(* CODESYS project sensata_laser.library
   Company: Sensata Technologies
   DocFormat: reStructuredText
   Description: This library is for the Laser devices
   Version: 1.0.1
   Placeholder: Sensata_Laser
   Title: Sensata_Laser

Project tree, tasks and I/O mapping:
  libraries: Sensata_Common, * (Sensata Technologies); Sensata_Utilities, * (Sensata Technologies); Tc2_Standard, * (Beckhoff Automation GmbH); Tc2_System, * (Beckhoff Automation GmbH); Tc2_Utilities, * (Beckhoff Automation GmbH); Tc3_Module, * (Beckhoff Automation GmbH)
  Abstract/
    function block FB_Laser [ST]: M_GetLaserStatus, M_LaserOff, M_LaserOn, P_bLaserControlBusy, P_bLaserOn
    function block FB_LaserMarker [ST]: M_SendMarkingParams_BlockRange, M_StartMarking, M_StopMarking, M_UpdateAllMarkingInformation, M_UpdateSingleBlockMarkingInformation, M_GetLaserStatus
    function block FB_LaserScanner [ST]: M_Trigger
  Concrete/
    IPG/
      function block FB_IPGD30 [ST]: M_Abort, P_bAbortBusy, M_Connect, M_Disconnect, M_GetConnectStatus, P_bConnectBusy, P_bConnected, M_Disable, M_Enable, M_GetEnableStatus, P_bEnableBusy, P_bEnabled, M_GetPowerStatus, M_PowerOff, M_PowerOn, P_bPowerBusy, P_bPoweredOn, M_GetCurrentProgram, M_GetProgramState, M_LoadProgram, M_PauseProgram, M_StartProgram, M_StopProgram, P_bProgramControlBusy, P_enumProgramState, P_strCurrentProgram, M_Reset, P_bResetBusy, A_CommandRecovery, M_RouterHelper
      function block FB_IPGWeld [ST]: M_Abort, P_bAbortBusy, M_Connect, M_Disconnect, M_GetConnectStatus, P_bConnectBusy, P_bConnected, M_Disable, M_Enable, M_GetEnableStatus, P_bEnableBusy, P_bEnabled, M_GetPowerStatus, M_PowerOff, M_PowerOn, P_bPowerBusy, P_bPoweredOn, M_GetCurrentProgram, M_GetProgramState, M_LoadProgram, M_PauseProgram, M_StartProgram, M_StopProgram, P_bProgramControlBusy, P_enumProgramState, P_strCurrentProgram, M_Reset, P_bResetBusy, M_Trigger, A_CommandRecovery, M_CommandTemplate, M_RouterHelper
    Keyence MDX-2000/
      function block FB_KeyenceLaserMarkerMDX2000 [LD]: M_Connect, M_Disconnect, M_GetConnectStatus, P_bConnectBusy, P_bConnected, M_PeakCurrentProgram, M_SendMarkingParams_BlockRange, M_StartMarking, M_StopMarking, M_UpdateAllMarkingInformation, M_UpdateSingleBlockMarkingInformation, M_GetCurrentProgram, M_GetProgramState, M_LoadProgram, M_PauseProgram, M_SaveCurrentLaserProgramtoPC, M_SendProgramtoLaser, M_StartProgram, M_StopProgram, M_UpdateSingleProgramBlockData, M_UpdateSingleProgramBlockMarkEnabled, P_bProgramControlBusy, P_enumProgramState, P_strCurrentProgram, M_GetLaserActivatedStatus, M_GetLaserErrorStatus, M_GetLaserMarkingStatus, M_GetLaserStatus, M_Reset, P_bResetBusy, A_CommandRecovery, M_RouterHelper
      data type KeyenceLaserMarkerMDX2000_Error
  DUTs/
    data type BlockTypes
    data type OneBlockInfo
  Interfaces/
    interface I_LaserControl: M_GetLaserStatus, M_LaserOff, M_LaserOn, P_bLaserControlBusy, P_bLaserOn
    interface I_Markable: M_StartMarking, M_StopMarking, M_UpdateAllMarkingInformation, M_UpdateSingleBlockMarkingInformation
    interface I_Triggerable: M_Trigger
  Project Information/
    function F_GetCompany [ST]
    function F_GetTitle [ST]
    function F_GetVersion [ST]
  Version/
    global variables Global_Version
  global variables GVL_LaserMarker
*)

// Concrete/Keyence MDX-2000/KeyenceLaserMarkerMDX2000_Error
{attribute 'qualified_only'}
{attribute 'strict'}
TYPE KeyenceLaserMarkerMDX2000_Error :
(
	None := 0,
	
	CommandRouterError							:= 0100, 		// Error on the command router FB
	CommandFault 								:= 0101, 		// Command failed to execute
	                            				         		
	FailedToConnect 							:= 0200, 		// Connect command failed
	FailedToDisconnect 							:= 0201, 		// Disonnect command failed
	FailedToGetConnectStatus 					:= 0202, 		// GetConnectStatus command failed
	                                                     		
	FailedToPeakCurrentProgram  				:= 0300, 		// Failed to Peak Current Program 
	FailedToSaveCurrentLaserProgramToPC 		:= 0301, 		//Failed to Save Current Laser Program to PC
	FailedToSendProgramToLaser					:= 0302, 		// Failed to Send Program To Laser
	FailedToStartMarking						:= 0303, 		// Laser Failed to Start Marking
	FailedToStopMarking							:= 0304, 		// Laser Failed to Stop Marking
	FailedToLoadProgram							:= 0310, 		// LoadProgram command failed
	FailedToGetCurrentProgram					:= 0311, 		// GetCurrentProgram command failed
	FailedToStartProgram						:= 0312, 		// StartProgram command failed
	FailedToStopProgram							:= 0313, 		// StopProgram command failed
	FailedToPauseProgram						:= 0314, 		// PauseProgram command failed
	FailedToGetProgramState						:= 0315, 		// GetProgramState command failed
	FailedToGetLaserStatus						:= 0316, 		// GetLaserStatus command failed
	FailedToGetLaserErrorStatus 				:= 0317, 		// GetLaserErrorStatus command failed
	FailedToGetLaserMarkingStatus 				:= 0318, 		// GetLaserMarkingStatus command failed
	FailedToGetLaserActivatedStatus				:= 0319, 		// GetLaserActivatedStatus command failed
	FailedToUpdateSingleBlockMarkEnabledProperty := 0320,		// UpdateSingleBlockMarkEnabled command failed
	FailedToUpdateSingleBlockData				:= 0321,		// UpdateSingleBlockData command failed
	FailedToUpdateAllMarkingInformation			:= 0322,		// UpdateAllMarkingInformation command failed
	FailedToUpdateSingleBlockMarkingInformation := 0323,		// UpdateSingleBlockMarkingInformation command failed
	FailedToGetPartLimitsFromDB					:= 0324,		// GetPartLimitsFromDB command failed
	FailedToSendMarkingParams_BlockRange        := 0325,		// SendMarkingParams_BlockRange command failed
                                                     		
	FailedToEnable								:= 0400, 		// Enable command failed
	FailedToDisable								:= 0401, 		// Disable command failed
	FailedToGetEnableStatus						:= 0402, 		// GetEnableStatus command failed
	                            				         		
	FailedToPowerOn								:= 0500, 		// PowerOn command failed
	FailedToPowerOff							:= 0501, 		// PowerOff command failed
	FailedToGetPowerStatus						:= 0502, 		// GetPowerStatus command failed
	                            				         		
	FailedToReset								:= 0600, 		// Reset command failed
	FailedToClearLaserErrors					:= 0601, 		// Failed to Clear Laser Errors
                                				         		
	FailedToGetSafetyStatus						:= 0700, 		// GetSafetyStatus command failed
	RobotSafetyFault							:= 0701  		// Robot safety fault occurred
) UDINT;
END_TYPE

// DUTs/BlockTypes
{attribute 'qualified_only'}
{attribute 'strict'}
TYPE BlockTypes :
(
  BLOCK_CHARACTER:=0, 
  BLOCK_RESERVED1:=1, 
  BLOCK_BARCODE:=2, 
  BLOCK_GS1DATABAR:=3, 
  BLOCK_2DCODE:=4, 
  BLOCK_RESERVED2:=5, 
  BLOCK_LOGO:=6, 
  BLOCK_PHOTO:=7, 
  BLOCK_PROCESSING:=8, 
  BLOCK_RESERVED3:=9
)INT;
END_TYPE

// DUTs/OneBlockInfo
TYPE OneBlockInfo :
STRUCT
	MarkEnabled : BOOL;
	BlockText : T_MaxString;
END_STRUCT
END_TYPE

// Version/Global_Version
{attribute 'TcGenerated'}
{attribute 'no-analysis'}
{attribute 'linkalways'}
// This function has been automatically generated from the project information.
VAR_GLOBAL CONSTANT
	{attribute 'const_non_replaced'}
	stLibVersion_Sensata_Laser : ST_LibVersion := (iMajor := 1, iMinor := 0, iBuild := 1, iRevision := 0, nFlags := 0, sVersion := '1.0.1');
END_VAR

// GVL_LaserMarker
VAR_GLOBAL
	LaserConnected : BOOL := FALSE;
	LaserDisconnected : BOOL := FALSE;
	LaserMarkerErrorsCleared : BOOL := FALSE;
	UpdateAllBlocksInLaserProgramSuccess : BOOL := FALSE;
	UpdateSingleBlockInLaserProgramSuccess : BOOL := FALSE;
	UpdateSingleBlockMarkEnabledSuccess : BOOL := FALSE;
	PeakCurrentProgramSuccess : BOOL := FALSE;
	SendProgramToLaserSuccess : BOOL := FALSE;
	SaveCurrentLaserProgramToPCSuccess : BOOL := FALSE;
	StartMarkingSuccess : BOOL := FALSE;
	StopMarkingSuccess : BOOL := FALSE;
	_bIsLaserActivated : BOOL := FALSE;
	_bIsLaserError : BOOL := FALSE;
	_bIsLaserMarking : BOOL := FALSE;
	KeyenceLaserProgramFolder : STRING := 'C:\MSDCommon\MarkingFiles\Program';
	KeyenceLaserModel : STRING := 'MARKINGUNIT_MDX2520';//For Marker Builder Plus and HVC(APT inline Cal #31) DAGZ181089
	KeyenceLaserIPAddress : STRING := '127.0.0.1';

END_VAR

// Abstract/FB_Laser
FUNCTION_BLOCK FB_Laser EXTENDS FB_Device IMPLEMENTS
I_LaserControl
VAR_INPUT
END_VAR
VAR_OUTPUT
END_VAR
VAR
	dev_bLaserOn: BOOL; // TRUE if the laser is on
END_VAR


METHOD M_GetLaserStatus : BOOL
VAR_OUTPUT
	(* TRUE if the laser is on, FALSE otherwise. *)
	bLaserOn	: BOOL;
END_VAR
bLaserOn:=dev_bLaserOn;
M_GetLaserStatus:=TRUE;
END_METHOD

(*Turn off Laser*)

METHOD M_LaserOff : BOOL
dev_bLaserOn:=FALSE;
M_LaserOff := TRUE;
THIS^.M_LogWarning('M_LaserOff is not implemented!');
END_METHOD

(*Turn On Laser*)
METHOD M_LaserOn : BOOL
dev_bLaserOn:=TRUE;
M_LaserOn := TRUE;
THIS^.M_LogWarning('M_LaserOn is not implemented!');
END_METHOD


(* This property should be TRUE while any method in this interface is actively
	executing, or FALSE otherwise. *)
PROPERTY P_bLaserControlBusy : BOOL
GET
P_bLaserControlBusy := FALSE;
END_GET
END_PROPERTY


(* This should be set to TRUE if M_LaserOn is successful or M_GetLaserStatus
	determines the laser to be On, and set to FALSE if M_LaserOff is
	called at all, M_GetLaserStatus fails, or M_GetLaserStatus determines
	the laser to be not on. *)
PROPERTY P_bLaserOn : BOOL
GET
P_bLaserOn:=dev_bLaserOn;
END_GET
END_PROPERTY

END_FUNCTION_BLOCK

// Interfaces/I_LaserControl
INTERFACE I_LaserControl

METHOD M_GetLaserStatus : BOOL
VAR_INPUT
END_VAR
VAR_OUTPUT
   	(* TRUE if the laser is on, FALSE otherwise. *)
	bLaserOn	: BOOL;
END_VAR
END_METHOD

METHOD M_LaserOff : BOOL
VAR_INPUT
END_VAR
END_METHOD

METHOD M_LaserOn : BOOL
VAR_INPUT
END_VAR
END_METHOD

(* This property should be TRUE while any method in this interface is actively
	executing, or FALSE otherwise. *)
PROPERTY P_bLaserControlBusy : BOOL
GET
END_GET
END_PROPERTY

(* This should be set to TRUE if M_LaserOn is successful or M_GetLaserStatus
	determines the laser to be On, and set to FALSE if M_LaserOff is
	called at all, M_GetLaserStatus fails, or M_GetLaserStatus determines
	the laser to be not on. *)
PROPERTY P_bLaserOn : BOOL
GET
END_GET
END_PROPERTY

END_INTERFACE

// Abstract/FB_LaserMarker
FUNCTION_BLOCK ABSTRACT FB_LaserMarker EXTENDS FB_Device IMPLEMENTS 
		I_Markable
VAR_INPUT
	//Send Marking Parameters Block Range
	in_PartNoStart : INT;//Part No Start
	in_PartNoEnd : INT;//Part No End
	in_BlockRangeData : T_MaxString;// The data compiled for blocks between Start Number and End Number mentioned
END_VAR
VAR_OUTPUT
END_VAR
VAR
END_VAR

METHOD PUBLIC M_SendMarkingParams_BlockRange : BOOL
VAR_INPUT
//	in_Data : T_MaxString;
//	in_PartNoStart : INT;
//	in_PartNoEnd : INT;
	in_MarkEnabled : BOOL;
END_VAR

VAR CONSTANT
	_strCOMMAND_NAME : T_MaxString	:= 'SendMarkingParams_BlockRange'; // Name of the API method
	_timeCOMMAND_TIMEOUT : TIME		:= T#30S; // Max time to receive API response
	_strSTART_MSG : T_MaxString		:= 'SendingMarkingParamsforBlockRange'; // Prints when method starts
	_strEND_MSG : T_MaxString		:= 'SentMarkingParamsforBlockRange'; // Prints when method finishes
	_udintERROR_ID : UDINT			:= KeyenceLaserMarkerMDX2000_Error.FailedToSendMarkingParams_BlockRange; // Error ID to set if command fails
	_strERROR_MSG : T_MaxString		:= 'Failed to send marking params for Block Range!'; // Error message to set if command fails
END_VAR

VAR_INST
	_inst_arrParams: T_ApiParameterList; // Parameters array
	_inst_arrOutputs: T_ApiParameterList; // Outputs array
	_inst_strRet: T_ApiParamValue; // Return string from the router
	_inst_intStep: INT; // Current method step
	_inst_fbParams: FB_ApiParamBuilder; // Parameter builder FB
END_VAR

VAR
	_bComplete: BOOL; // True if the routing finishes
	_intRet: INT; // Return string converted to an integer
	_bResult : BOOL; // Output of the method
END_VAR
M_SendMarkingParams_BlockRange := TRUE;
THIS^.M_LogWarning('M_SendMarkingParams_BlockRange is not implemented!');
END_METHOD

METHOD M_StartMarking : BOOL
M_StartMarking := TRUE;
THIS^.M_LogWarning('M_StartMarking is not implemented!');
END_METHOD

METHOD M_StopMarking : BOOL
M_StopMarking := TRUE;
THIS^.M_LogWarning('StopMarking is not implemented!');
END_METHOD

METHOD M_UpdateAllMarkingInformation : BOOL
VAR_INPUT
	MaxNumberOfBlocks	: INT;
//	MarkingInfo_Array	: ARRAY [0..255] OF OneBlockInfo;
END_VAR
M_UpdateAllMarkingInformation := TRUE;
THIS^.M_LogWarning('M_UpdateAllMarkingInformation is not implemented!');
END_METHOD

METHOD PUBLIC M_UpdateSingleBlockMarkingInformation : BOOL
VAR_INPUT
	BlockNumber : INT;
	BlockData : STRING;
	MarkEnabled : BOOL;
END_VAR
M_UpdateSingleBlockMarkingInformation := TRUE;
THIS^.M_LogWarning('M_UpdateSingleBlockMarkingInformation is not implemented!');
END_METHOD

METHOD PUBLIC ABSTRACT M_GetLaserStatus : BOOL
VAR_INPUT
END_VAR
VAR_OUTPUT
	out_string_laserStatus : STRING;
END_VAR
//M_GetLaserStatus := TRUE;
//THIS^.M_LogWarning('M_GetLaserStatus is not implemented!');
END_METHOD

END_FUNCTION_BLOCK

// Interfaces/I_Markable
INTERFACE I_Markable

METHOD M_StartMarking : BOOL
VAR_INPUT
END_VAR
END_METHOD

METHOD M_StopMarking : BOOL
VAR_INPUT
END_VAR
END_METHOD

METHOD M_UpdateAllMarkingInformation : BOOL
VAR_INPUT
	MaxNumberOfBlocks	: INT;
//	MarkingInfo_Array	: ARRAY [0..255] OF OneBlockInfo;//Commenting this because this might not be needed incase data is flowing from DB table to C# class itself instead of 
														 //going through the C# to beckhoff to C# 
END_VAR
END_METHOD

METHOD M_UpdateSingleBlockMarkingInformation : BOOL
VAR_INPUT
	BlockNumber : INT;
	BlockData : STRING;
	MarkEnabled : BOOL;
END_VAR
END_METHOD

END_INTERFACE

// Abstract/FB_LaserScanner
FUNCTION_BLOCK FB_LaserScanner EXTENDS FB_Device IMPLEMENTS I_Triggerable
VAR_INPUT
END_VAR
VAR_OUTPUT
END_VAR
VAR
END_VAR

(* Triggers an action from a laser scanner such as marking, welding, cleaning, etc. *)
METHOD M_Trigger : BOOL
THIS^.M_LogWarning('M_Trigger not implemented!');
M_Trigger := TRUE;
END_METHOD

END_FUNCTION_BLOCK

// Interfaces/I_Triggerable
INTERFACE I_Triggerable

(* Triggers an action from a laser scanner such as marking, welding, cleaning, etc. *)
METHOD M_Trigger : BOOL
VAR_INPUT
END_VAR
END_METHOD

END_INTERFACE

// Concrete/IPG/FB_IPGD30
(*
	Function block for controlling the Wobble controller IPG D30 from the API
*)
FUNCTION_BLOCK FB_IPGD30 EXTENDS FB_LaserScanner
	IMPLEMENTS 
		I_Abortable,
		I_Connectable, 
		I_Powerable,
		I_Enableable,
		I_Resettable,
		I_Programmable
VAR_INPUT
	(* Reference to an FB_CommandRouter function block to send commands
		to a command router in the API. *)
	in_fbApi : REFERENCE TO FB_CommandRouter;
	(* ID of the API module to send router commands to. *)
	in_strApiModuleId: T_MaxString;
	
	(*program num to load - Program numbers from 0 to 6*)
	in_intProgramNum:INT;
	(*Wobble pattern :number 0 to 4 for wobble type;
	0 Wobble Mode - Clockwise Circle;
	1 Wobble Mode - Counter Clockwise Circle;
	2 Wobble Mode - Linear;
	3 Wobble Mode - Figure 8 ;
	4 Wobble Mode - Infinity
 	*)
	in_intWobbleMode:INT;
	(*Wobble Frquency*)
	in_intWobbleFreq:INT;
	(*Wobble Amplitude*)
	in_lrWobbleAmp:LREAL;
	(*Wobble offset*)
	in_intWobbleOffset:INT;
	(*Material speed; minimum 1 *)
	in_intMaterialSpeed:INT:=1;
	(*Save; minimum 1 *)
	in_intSaveSetting:INT;
END_VAR
VAR_IN_OUT
END_VAR
VAR_OUTPUT
END_VAR
VAR CONSTANT
END_VAR
VAR
	bConnected: BOOL; // Value of P_bConnected
	bEnabled: BOOL; // Value of P_bEnabled
	bPoweredOn: BOOL; // Value of P_bPoweredOn
	strLoadedProgram: STRING(255); // Value of P_strLoadedProgram
	enumProgramState: E_PROGRAMSTATE; // Value of P_enumProgramState
	
	bRouterBusy: BOOL; // TRUE while M_RouterHelper is being used by a method

	bTemplateBusy: BOOL;
	bConnectBusy: BOOL;
	bDisconnectBusy: BOOL;
	bGetConnectStatusBusy: BOOL;
	bEnableBusy: BOOL;
	bDisableBusy: BOOL;
	bGetEnableStatusBusy: BOOL;
	bPowerOnBusy: BOOL;
	bPowerOffBusy: BOOL;
	bGetPowerStatusBusy: BOOL;
	bGetCurrentProgramBusy: BOOL;
	bGetProgramStateBusy: BOOL;
	bLoadProgramBusy: BOOL;
	bPauseProgramBusy: BOOL;
	bStartProgramBusy: BOOL;
	bStopProgramBusy: BOOL;
	bResetBusy: BOOL;
	bAbortBusy: BOOL;
	bRouterHelperBusy: BOOL;
	
	intTemplateStep: INT;
	intConnectStep: INT;
	intDisconnectStep: INT;
	intGetConnectStatusStep: INT;
	intEnableStep: INT;
	intDisableStep: INT;
	intGetEnableStatusStep: INT;
	intPowerOnStep: INT;
	intPowerOffStep: INT;
	intGetCurrentProgramStep: INT;
	intGetProgramStateStep: INT;
	intLoadProgramStep: INT;
	intPauseProgramStep: INT;
	intStartProgramStep: INT;
	intStopProgramStep: INT;
	intResetStep: INT;
	intAbortStep: INT;
	intGetPowerStatusStep: INT;
	intRouterHelperStep: INT;
END_VAR

A_CommandRecovery();

(* This method should establish any external connections required to use the
	functions of the device, and return TRUE and set P_bConnected to TRUE once
	connected. *)
METHOD M_Abort : BOOL
VAR CONSTANT
	_strCOMMAND_NAME : T_MaxString	:= 'Abort'; // Name of the API method
	_timeCOMMAND_TIMEOUT : TIME		:= T#30S; // Max time to receive API response
	_strSTART_MSG : T_MaxString		:= 'Aborting'; // Prints when method starts
	_strEND_MSG : T_MaxString		:= 'Aborted'; // Prints when method finishes
	_udintERROR_ID : UDINT			:= E_ApiDeviceError.FailedToAbort; // Error ID to set if command fails
	_strERROR_MSG : T_MaxString		:= 'Abort failed!'; // Error message to set if command fails
END_VAR
VAR_INST
	_inst_arrParams: T_ApiParameterList; // Parameters array
	_inst_arrOutputs: T_ApiParameterList; // Outputs array
	_inst_strRet: T_ApiParamValue; // Return string from the router
	_inst_intStep: INT; // Current method step
	_inst_fbParams: FB_ApiParamBuilder; // Parameter builder FB
END_VAR
VAR
	_bComplete: BOOL; // True if the routing finishes
	_intRet: INT; // Return string converted to an integer
	_bResult : BOOL; // Output of the method
	_pArgs: PVOID; // Arguments pointer
END_VAR
_bResult := FALSE;

// Recover from premature stop
bAbortBusy := TRUE;
_inst_intStep := intAbortStep;

// Steps
(* TEMPLATE: Parameters should be added in step 10, and output
	parsing should be added in step 30. *)
CASE _inst_intStep OF
	0: // Wait for no error and router not busy
		IF NOT THIS^.P_bError AND NOT bRouterBusy THEN
			bRouterBusy := TRUE;
			_inst_intStep := _inst_intStep + 10;
		END_IF
		
	10: // Initialize parameters
		THIS^.M_LogMessage(_strSTART_MSG);
		_inst_fbParams.M_ClearParameters();
		_pArgs := _inst_fbParams.M_AddEmptyStruct('args');
		// TEMPLATE: Add any parameters here
		_inst_fbParams.M_OutputToParameterList(_inst_arrParams);
		_inst_intStep := _inst_intStep + 10;
		
	20: // Route the command
		_bComplete := M_RouterHelper(
			_in_strMethodName := _strCOMMAND_NAME, 
			_in_timeTimeout := _timeCOMMAND_TIMEOUT,
			_inout_arrParams := _inst_arrParams,
			_inout_arrOutputs := _inst_arrOutputs,
			_out_strReturnValue=>_inst_strRet);
		
		// If route completed, move to next step
		IF _bComplete THEN
			_inst_intStep := _inst_intStep + 10;
			bRouterBusy := FALSE;
		ELSIF THIS^.P_bError THEN
			_inst_intStep := 0;
			bRouterBusy := FALSE;
		END_IF
		
	30: // Parse results
		_intRet := STRING_TO_INT(_inst_strRet);
		IF _intRet > 0 THEN
			_bResult := TRUE;
			THIS^.M_LogMessage(_strEND_MSG);
			_inst_fbParams.M_LoadFromParameterList(_inst_arrOutputs);
			// TEMPLATE: Do any parsing here
			
		// Set error if command failed
		ELSE
			THIS^.M_SetError(_udintERROR_ID, _strERROR_MSG);
		END_IF
		
		// Go back to start
		_inst_intStep := 0;
END_CASE

M_Abort := _bResult;
intAbortStep := _inst_intStep;
END_METHOD

(* This property should be TRUE while any method in this interface is actively
	executing, or FALSE otherwise. *)
PROPERTY P_bAbortBusy : BOOL
GET
P_bAbortBusy := bRouterBusy;
END_GET
END_PROPERTY

(* This method should establish any external connections required to use the
	functions of the device, and return TRUE and set P_bConnected to TRUE once
	connected. *)
METHOD M_Connect : BOOL
VAR CONSTANT
	_strCOMMAND_NAME : T_MaxString	:= 'Connect'; // Name of the API method
	_timeCOMMAND_TIMEOUT : TIME		:= T#30S; // Max time to receive API response
	_strSTART_MSG : T_MaxString		:= 'Connecting'; // Prints when method starts
	_strEND_MSG : T_MaxString		:= 'Connected'; // Prints when method finishes
	_udintERROR_ID : UDINT			:= E_ApiDeviceError.FailedToConnect; // Error ID to set if command fails
	_strERROR_MSG : T_MaxString		:= 'Failed to connect!'; // Error message to set if command fails
END_VAR
VAR_INST
	_inst_arrParams: T_ApiParameterList; // Parameters array
	_inst_arrOutputs: T_ApiParameterList; // Outputs array
	_inst_strRet: T_ApiParamValue; // Return string from the router
	_inst_intStep: INT; // Current method step
	_inst_fbParams: FB_ApiParamBuilder; // Parameter builder FB
END_VAR
VAR
	_bComplete: BOOL; // True if the routing finishes
	_intRet: INT; // Return string converted to an integer
	_bResult : BOOL; // Output of the method
	_pArgs: PVOID; // Arguments pointer
END_VAR
_bResult := FALSE;

// Recover from premature stop
bConnectBusy := TRUE;
_inst_intStep := intConnectStep;

// Steps
(* TEMPLATE: Parameters should be added in step 10, and output
	parsing should be added in step 30. *)
CASE _inst_intStep OF
	0: // Wait for no error and router not busy
		IF NOT THIS^.P_bError AND NOT bRouterBusy THEN
			bRouterBusy := TRUE;
			_inst_intStep := _inst_intStep + 10;
		END_IF
		
	10: // Initialize parameters
		THIS^.M_LogMessage(_strSTART_MSG);
		_inst_fbParams.M_ClearParameters();
		_pArgs := _inst_fbParams.M_AddEmptyStruct('args');
		// TEMPLATE: Add any parameters here
		_inst_fbParams.M_OutputToParameterList(_inst_arrParams);
		_inst_intStep := _inst_intStep + 10;
		
	20: // Route the command
		_bComplete := M_RouterHelper(
			_in_strMethodName := _strCOMMAND_NAME, 
			_in_timeTimeout := _timeCOMMAND_TIMEOUT,
			_inout_arrParams := _inst_arrParams,
			_inout_arrOutputs := _inst_arrOutputs,
			_out_strReturnValue=>_inst_strRet);
		
		// If route completed, move to next step
		IF _bComplete THEN
			_inst_intStep := _inst_intStep + 10;
			bRouterBusy := FALSE;
		ELSIF THIS^.P_bError THEN
			_inst_intStep := 0;
			bRouterBusy := FALSE;
		END_IF
		
	30: // Parse results
		_intRet := STRING_TO_INT(_inst_strRet);
		IF _intRet > 0 THEN
			_bResult := TRUE;
			THIS^.M_LogMessage(_strEND_MSG);
			_inst_fbParams.M_LoadFromParameterList(_inst_arrOutputs);
			// TEMPLATE: Do any parsing here
			bConnected := TRUE;
			
		// Set error if command failed
		ELSE
			THIS^.M_SetError(_udintERROR_ID, _strERROR_MSG);
		END_IF
		
		// Go back to start
		_inst_intStep := 0;
END_CASE

M_Connect := _bResult;
intConnectStep := _inst_intStep;
END_METHOD

(* This method should break any connections established by M_Connect. It should
	immediately set P_bConnected to false unless all connections are known to
	be still active, and return TRUE once those connections are all fully
	disconnected. *)
METHOD M_Disconnect : BOOL
VAR CONSTANT
	_strCOMMAND_NAME : T_MaxString	:= 'Disconnect'; // Name of the API method
	_timeCOMMAND_TIMEOUT : TIME		:= T#30S; // Max time to receive API response
	_strSTART_MSG : T_MaxString		:= 'Disconnecting'; // Prints when method starts
	_strEND_MSG : T_MaxString		:= 'Disconnected'; // Prints when method finishes
	_udintERROR_ID : UDINT			:= E_ApiDeviceError.FailedToDisconnect; // Error ID to set if command fails
	_strERROR_MSG : T_MaxString		:= 'Failed to disconnect!'; // Error message to set if command fails
END_VAR
VAR_INST
	_inst_arrParams: T_ApiParameterList; // Parameters array
	_inst_arrOutputs: T_ApiParameterList; // Outputs array
	_inst_strRet: T_ApiParamValue; // Return string from the router
	_inst_intStep: INT; // Current method step
	_inst_fbParams: FB_ApiParamBuilder; // Parameter builder FB
END_VAR
VAR
	_bComplete: BOOL; // True if the routing finishes
	_intRet: INT; // Return string converted to an integer
	_bResult : BOOL; // Output of the method
	_pArgs: PVOID; // Arguments pointer
END_VAR
_bResult := FALSE;

// Recover from premature stop
bDisconnectBusy := TRUE;
_inst_intStep := intDisconnectStep;

// Steps
(* TEMPLATE: Parameters should be added in step 10, and output
	parsing should be added in step 30. *)
CASE _inst_intStep OF
	0: // Wait for no error and router not busy
		IF NOT THIS^.P_bError AND NOT bRouterBusy THEN
			bRouterBusy := TRUE;
			_inst_intStep := _inst_intStep + 10;
		END_IF
		
	10: // Initialize parameters
		THIS^.M_LogMessage(_strSTART_MSG);
		_inst_fbParams.M_ClearParameters();
		_pArgs := _inst_fbParams.M_AddEmptyStruct('args');
		// TEMPLATE: Add any parameters here
		_inst_fbParams.M_OutputToParameterList(_inst_arrParams);
		_inst_intStep := _inst_intStep + 10;
		
	20: // Route the command
		_bComplete := M_RouterHelper(
			_in_strMethodName := _strCOMMAND_NAME, 
			_in_timeTimeout := _timeCOMMAND_TIMEOUT,
			_inout_arrParams := _inst_arrParams,
			_inout_arrOutputs := _inst_arrOutputs,
			_out_strReturnValue=>_inst_strRet);
		
		// If route completed, move to next step
		IF _bComplete THEN
			_inst_intStep := _inst_intStep + 10;
			bRouterBusy := FALSE;
		ELSIF THIS^.P_bError THEN
			_inst_intStep := 0;
			bRouterBusy := FALSE;
		END_IF
		
	30: // Parse results
		_intRet := STRING_TO_INT(_inst_strRet);
		IF _intRet > 0 THEN
			_bResult := TRUE;
			THIS^.M_LogMessage(_strEND_MSG);
			_inst_fbParams.M_LoadFromParameterList(_inst_arrOutputs);
			// TEMPLATE: Do any parsing here
			bConnected := FALSE;
			
		// Set error if command failed
		ELSE
			THIS^.M_SetError(_udintERROR_ID, _strERROR_MSG);
		END_IF
		
		// Go back to start
		_inst_intStep := 0;
END_CASE

M_Disconnect := _bResult;
intDisconnectStep := _inst_intStep;
END_METHOD

(* This method should explicitly check the connection status of the device.
	Once the connection status is known, this method should return TRUE.
	If this method fails, P_bConnected should be set to FALSE since the device
	is not absolutely known to still be connected. *)
METHOD M_GetConnectStatus : BOOL
VAR_OUTPUT
	(* This should return TRUE if all connections required to make the device
		function properly are known to be connected, and FALSE otherwise. *)
	bConnected	: BOOL;
END_VAR
VAR CONSTANT
	_strCOMMAND_NAME : T_MaxString	:= 'GetConnectStatus'; // Name of the API method
	_timeCOMMAND_TIMEOUT : TIME		:= T#5S; // Max time to receive API response
	_strSTART_MSG : T_MaxString		:= 'Getting connection status'; // Prints when method starts
	_strEND_MSG : T_MaxString		:= 'Received connection status'; // Prints when method finishes
	_udintERROR_ID : UDINT			:= E_ApiDeviceError.FailedToGetConnectStatus; // Error ID to set if command fails
	_strERROR_MSG : T_MaxString		:= 'Failed to get connection status!'; // Error message to set if command fails
END_VAR
VAR_INST
	_inst_arrParams: T_ApiParameterList; // Parameters array
	_inst_arrOutputs: T_ApiParameterList; // Outputs array
	_inst_strRet: T_ApiParamValue; // Return string from the router
	_inst_intStep: INT; // Current method step
	_inst_fbParams: FB_ApiParamBuilder; // Parameter builder FB
END_VAR
VAR
	_bComplete: BOOL; // True if the routing finishes
	_intRet: INT; // Return string converted to an integer
	_bResult : BOOL; // Output of the method
	_pArgs: PVOID; // Arguments pointer
END_VAR
_bResult := FALSE;

// Recover from premature stop
bGetConnectStatusBusy := TRUE;
_inst_intStep := intGetConnectStatusStep;

// Steps
(* TEMPLATE: Parameters should be added in step 10, and output
	parsing should be added in step 30. *)
CASE _inst_intStep OF
	0: // Wait for no error and router not busy
		IF NOT THIS^.P_bError AND NOT bRouterBusy THEN
			bRouterBusy := TRUE;
			_inst_intStep := _inst_intStep + 10;
		END_IF
		
	10: // Initialize parameters
		THIS^.M_LogMessage(_strSTART_MSG);
		_inst_fbParams.M_ClearParameters();
		_pArgs := _inst_fbParams.M_AddEmptyStruct('args');
		// TEMPLATE: Add any parameters here
		_inst_fbParams.M_OutputToParameterList(_inst_arrParams);
		_inst_intStep := _inst_intStep + 10;
		
	20: // Route the command
		_bComplete := M_RouterHelper(
			_in_strMethodName := _strCOMMAND_NAME, 
			_in_timeTimeout := _timeCOMMAND_TIMEOUT,
			_inout_arrParams := _inst_arrParams,
			_inout_arrOutputs := _inst_arrOutputs,
			_out_strReturnValue=>_inst_strRet);
		
		// If route completed, move to next step
		IF _bComplete THEN
			_inst_intStep := _inst_intStep + 10;
			bRouterBusy := FALSE;
		ELSIF THIS^.P_bError THEN
			_inst_intStep := 0;
			bRouterBusy := FALSE;
		END_IF
		
	30: // Parse results
		_intRet := STRING_TO_INT(_inst_strRet);
		IF _intRet > 0 THEN
			_bResult := TRUE;
			THIS^.M_LogMessage(_strEND_MSG);
			_inst_fbParams.M_LoadFromParameterList(_inst_arrOutputs);
			// TEMPLATE: Do any parsing here
			THIS^.bConnected := _inst_fbParams.M_ParseBool(
				_inst_fbParams.M_GetParameter('connected'));
			bConnected := THIS^.bConnected;
			
		// Set error if command failed
		ELSE
			THIS^.M_SetError(_udintERROR_ID, _strERROR_MSG);
		END_IF
		
		// Go back to start
		_inst_intStep := 0;
END_CASE

M_GetConnectStatus := _bResult;
intGetConnectStatusStep := _inst_intStep;
END_METHOD

(* This property should be TRUE while any method in this interface is actively
	executing, or FALSE otherwise. *)
PROPERTY P_bConnectBusy : BOOL
GET
P_bConnectBusy := bRouterBusy;
END_GET
END_PROPERTY

(* This should be set to TRUE if M_Connect is successful or M_GetConnectStatus
	determines the device to be connected, and set to FALSE if M_Disconnect is
	called at all, M_GetConnectStatus fails, or M_GetConnectStatus determines
	the device to be not connected. *)
PROPERTY P_bConnected : BOOL
GET
P_bConnected := bConnected;
END_GET
END_PROPERTY

(* This method should return to the device to the state it was prior to being
	enabled. P_bEnabled should be immediately set to false unless the status of
	the device is explicitly known to still be enabled. After being disabled,
	the device should typically be unable to perform process steps. Once
	successfully disabled, this method should return TRUE. *)
METHOD M_Disable : BOOL
VAR CONSTANT
	_strCOMMAND_NAME : T_MaxString	:= 'Disable'; // Name of the API method
	_timeCOMMAND_TIMEOUT : TIME		:= T#30S; // Max time to receive API response
	_strSTART_MSG : T_MaxString		:= 'Disabling'; // Prints when method starts
	_strEND_MSG : T_MaxString		:= 'Disabled'; // Prints when method finishes
	_udintERROR_ID : UDINT			:= E_ApiDeviceError.FailedToDisable; // Error ID to set if command fails
	_strERROR_MSG : T_MaxString		:= 'Failed to disable!'; // Error message to set if command fails
END_VAR
VAR_INST
	_inst_arrParams: T_ApiParameterList; // Parameters array
	_inst_arrOutputs: T_ApiParameterList; // Outputs array
	_inst_strRet: T_ApiParamValue; // Return string from the router
	_inst_intStep: INT; // Current method step
	_inst_fbParams: FB_ApiParamBuilder; // Parameter builder FB
END_VAR
VAR
	_bComplete: BOOL; // True if the routing finishes
	_intRet: INT; // Return string converted to an integer
	_bResult : BOOL; // Output of the method
	_pArgs: PVOID; // Arguments pointer
END_VAR
_bResult := FALSE;

// Recover from premature stop
bDisableBusy := TRUE;
_inst_intStep := intDisableStep;

// Steps
(* TEMPLATE: Parameters should be added in step 10, and output
	parsing should be added in step 30. *)
CASE _inst_intStep OF
	0: // Wait for no error and router not busy
		IF NOT THIS^.P_bError AND NOT bRouterBusy THEN
			bRouterBusy := TRUE;
			_inst_intStep := _inst_intStep + 10;
		END_IF
		
	10: // Initialize parameters
		THIS^.M_LogMessage(_strSTART_MSG);
		_inst_fbParams.M_ClearParameters();
		_pArgs := _inst_fbParams.M_AddEmptyStruct('args');
		// TEMPLATE: Add any parameters here
		_inst_fbParams.M_OutputToParameterList(_inst_arrParams);
		_inst_intStep := _inst_intStep + 10;
		
	20: // Route the command
		_bComplete := M_RouterHelper(
			_in_strMethodName := _strCOMMAND_NAME, 
			_in_timeTimeout := _timeCOMMAND_TIMEOUT,
			_inout_arrParams := _inst_arrParams,
			_inout_arrOutputs := _inst_arrOutputs,
			_out_strReturnValue=>_inst_strRet);
		
		// If route completed, move to next step
		IF _bComplete THEN
			_inst_intStep := _inst_intStep + 10;
			bRouterBusy := FALSE;
		ELSIF THIS^.P_bError THEN
			_inst_intStep := 0;
			bRouterBusy := FALSE;
		END_IF
		
	30: // Parse results
		_intRet := STRING_TO_INT(_inst_strRet);
		IF _intRet > 0 THEN
			_bResult := TRUE;
			THIS^.M_LogMessage(_strEND_MSG);
			_inst_fbParams.M_LoadFromParameterList(_inst_arrOutputs);
			// TEMPLATE: Do any parsing here
			bEnabled := FALSE;
			
		// Set error if command failed
		ELSE
			THIS^.M_SetError(_udintERROR_ID, _strERROR_MSG);
		END_IF
		
		// Go back to start
		_inst_intStep := 0;
END_CASE

M_Disable := _bResult;
intDisableStep := _inst_intStep;
END_METHOD

(* This method should perform any tasks that must be performed after a device
	is energized, but prior to the device being used in a process, and then
	return TRUE and set P_bEnabled to TRUE once those tasks are completed. *)
METHOD M_Enable : BOOL
VAR CONSTANT
	_strCOMMAND_NAME : T_MaxString	:= 'Enable'; // Name of the API method
	_timeCOMMAND_TIMEOUT : TIME		:= T#30S; // Max time to receive API response
	_strSTART_MSG : T_MaxString		:= 'Enabling'; // Prints when method starts
	_strEND_MSG : T_MaxString		:= 'Enabled'; // Prints when method finishes
	_udintERROR_ID : UDINT			:= E_ApiDeviceError.FailedToEnable; // Error ID to set if command fails
	_strERROR_MSG : T_MaxString		:= 'Failed to enable!'; // Error message to set if command fails
END_VAR
VAR_INST
	_inst_arrParams: T_ApiParameterList; // Parameters array
	_inst_arrOutputs: T_ApiParameterList; // Outputs array
	_inst_strRet: T_ApiParamValue; // Return string from the router
	_inst_intStep: INT; // Current method step
	_inst_fbParams: FB_ApiParamBuilder; // Parameter builder FB
END_VAR
VAR
	_bComplete: BOOL; // True if the routing finishes
	_intRet: INT; // Return string converted to an integer
	_bResult : BOOL; // Output of the method
	_pArgs: PVOID; // Arguments pointer
END_VAR
_bResult := FALSE;

// Recover from premature stop
bEnableBusy := TRUE;
_inst_intStep := intEnableStep;

// Steps
(* TEMPLATE: Parameters should be added in step 10, and output
	parsing should be added in step 30. *)
CASE _inst_intStep OF
	0: // Wait for no error and router not busy
		IF NOT THIS^.P_bError AND NOT bRouterBusy THEN
			bRouterBusy := TRUE;
			_inst_intStep := _inst_intStep + 10;
		END_IF
		
	10: // Initialize parameters
		THIS^.M_LogMessage(_strSTART_MSG);
		_inst_fbParams.M_ClearParameters();
		_pArgs := _inst_fbParams.M_AddEmptyStruct('args');
		// TEMPLATE: Add any parameters here
		_inst_fbParams.M_OutputToParameterList(_inst_arrParams);
		_inst_intStep := _inst_intStep + 10;
		
	20: // Route the command
		_bComplete := M_RouterHelper(
			_in_strMethodName := _strCOMMAND_NAME, 
			_in_timeTimeout := _timeCOMMAND_TIMEOUT,
			_inout_arrParams := _inst_arrParams,
			_inout_arrOutputs := _inst_arrOutputs,
			_out_strReturnValue=>_inst_strRet);
		
		// If route completed, move to next step
		IF _bComplete THEN
			_inst_intStep := _inst_intStep + 10;
			bRouterBusy := FALSE;
		ELSIF THIS^.P_bError THEN
			_inst_intStep := 0;
			bRouterBusy := FALSE;
		END_IF
		
	30: // Parse results
		_intRet := STRING_TO_INT(_inst_strRet);
		IF _intRet > 0 THEN
			_bResult := TRUE;
			THIS^.M_LogMessage(_strEND_MSG);
			_inst_fbParams.M_LoadFromParameterList(_inst_arrOutputs);
			// TEMPLATE: Do any parsing here
			bEnabled := TRUE;
			
		// Set error if command failed
		ELSE
			THIS^.M_SetError(_udintERROR_ID, _strERROR_MSG);
		END_IF
		
		// Go back to start
		_inst_intStep := 0;
END_CASE

M_Enable := _bResult;
intEnableStep := _inst_intStep;
END_METHOD

(* This method should explicitly check the enable status of the device.
	Once the enable status is known, this method should return TRUE.
	If this method fails, P_bEnabled should be set to FALSE since the device
	is not absolutely known to still be enabled. *)
METHOD M_GetEnableStatus : BOOL
VAR_OUTPUT
	(* This should return TRUE if the device is explicitly known to be
		enabled, or FALSE otherwise. *)
	bEnabled	: BOOL;
END_VAR
VAR CONSTANT
	_strCOMMAND_NAME : T_MaxString	:= 'GetEnableStatus'; // Name of the API method
	_timeCOMMAND_TIMEOUT : TIME		:= T#5S; // Max time to receive API response
	_strSTART_MSG : T_MaxString		:= 'Getting enable status'; // Prints when method starts
	_strEND_MSG : T_MaxString		:= 'Received enable status'; // Prints when method finishes
	_udintERROR_ID : UDINT			:= E_ApiDeviceError.FailedToGetEnableStatus; // Error ID to set if command fails
	_strERROR_MSG : T_MaxString		:= 'Failed to get enable status!'; // Error message to set if command fails
END_VAR
VAR_INST
	_inst_arrParams: T_ApiParameterList; // Parameters array
	_inst_arrOutputs: T_ApiParameterList; // Outputs array
	_inst_strRet: T_ApiParamValue; // Return string from the router
	_inst_intStep: INT; // Current method step
	_inst_fbParams: FB_ApiParamBuilder; // Parameter builder FB
END_VAR
VAR
	_bComplete: BOOL; // True if the routing finishes
	_intRet: INT; // Return string converted to an integer
	_bResult : BOOL; // Output of the method
	_pArgs: PVOID; // Arguments pointer
END_VAR
_bResult := FALSE;

// Recover from premature stop
bGetEnableStatusBusy := TRUE;
_inst_intStep := intGetEnableStatusStep;

// Steps
(* TEMPLATE: Parameters should be added in step 10, and output
	parsing should be added in step 30. *)
CASE _inst_intStep OF
	0: // Wait for no error and router not busy
		IF NOT THIS^.P_bError AND NOT bRouterBusy THEN
			bRouterBusy := TRUE;
			_inst_intStep := _inst_intStep + 10;
		END_IF
		
	10: // Initialize parameters
		THIS^.M_LogMessage(_strSTART_MSG);
		_inst_fbParams.M_ClearParameters();
		_pArgs := _inst_fbParams.M_AddEmptyStruct('args');
		// TEMPLATE: Add any parameters here
		_inst_fbParams.M_OutputToParameterList(_inst_arrParams);
		_inst_intStep := _inst_intStep + 10;
		
	20: // Route the command
		_bComplete := M_RouterHelper(
			_in_strMethodName := _strCOMMAND_NAME, 
			_in_timeTimeout := _timeCOMMAND_TIMEOUT,
			_inout_arrParams := _inst_arrParams,
			_inout_arrOutputs := _inst_arrOutputs,
			_out_strReturnValue=>_inst_strRet);
		
		// If route completed, move to next step
		IF _bComplete THEN
			_inst_intStep := _inst_intStep + 10;
			bRouterBusy := FALSE;
		ELSIF THIS^.P_bError THEN
			_inst_intStep := 0;
			bRouterBusy := FALSE;
		END_IF
		
	30: // Parse results
		_intRet := STRING_TO_INT(_inst_strRet);
		IF _intRet > 0 THEN
			_bResult := TRUE;
			THIS^.M_LogMessage(_strEND_MSG);
			_inst_fbParams.M_LoadFromParameterList(_inst_arrOutputs);
			// TEMPLATE: Do any parsing here
			THIS^.bEnabled := _inst_fbParams.M_ParseBool(
				_inst_fbParams.M_GetParameter('enabled'));
			bEnabled := THIS^.bEnabled;
			
		// Set error if command failed
		ELSE
			THIS^.M_SetError(_udintERROR_ID, _strERROR_MSG);
		END_IF
		
		// Go back to start
		_inst_intStep := 0;
END_CASE

M_GetEnableStatus := _bResult;
intGetEnableStatusStep := _inst_intStep;
END_METHOD

(* This property should be TRUE while any method in this interface is actively
	executing, or FALSE otherwise. *)
PROPERTY P_bEnableBusy : BOOL
GET
P_bEnableBusy := bRouterBusy;
END_GET
END_PROPERTY

(* This should be set to TRUE if M_Enable is successful or M_GetEnableStatus
	determines the device to be enabled, and set to FALSE if M_Disable is
	called at all, M_GetEnableStatus fails, or M_GetEnableStatus determines
	the device to be not enabled. *)
PROPERTY P_bEnabled : BOOL
GET
P_bEnabled := bEnabled;
END_GET
END_PROPERTY

(* This method should explicitly check the power status of the device.
	Once the power status is known, this method should return TRUE.
	If this method fails, P_bPoweredOn should be set to FALSE since the device
	is not absolutely known to still be powered on. *)
METHOD M_GetPowerStatus : BOOL
VAR_OUTPUT
	(* This should return TRUE if the device is explicitly known to be
		powered on, or FALSE otherwise. *)
	bPoweredOn	: BOOL;
END_VAR
VAR CONSTANT
	_strCOMMAND_NAME : T_MaxString	:= 'GetPowerStatus'; // Name of the API method
	_timeCOMMAND_TIMEOUT : TIME		:= T#5S; // Max time to receive API response
	_strSTART_MSG : T_MaxString		:= 'Getting power status'; // Prints when method starts
	_strEND_MSG : T_MaxString		:= 'Received power status'; // Prints when method finishes
	_udintERROR_ID : UDINT			:= E_ApiDeviceError.FailedToGetPowerStatus; // Error ID to set if command fails
	_strERROR_MSG : T_MaxString		:= 'Failed to get power status!'; // Error message to set if command fails
END_VAR
VAR_INST
	_inst_arrParams: T_ApiParameterList; // Parameters array
	_inst_arrOutputs: T_ApiParameterList; // Outputs array
	_inst_strRet: T_ApiParamValue; // Return string from the router
	_inst_intStep: INT; // Current method step
	_inst_fbParams: FB_ApiParamBuilder; // Parameter builder FB
END_VAR
VAR
	_bComplete: BOOL; // True if the routing finishes
	_intRet: INT; // Return string converted to an integer
	_bResult : BOOL; // Output of the method
	_pArgs: PVOID; // Arguments pointer
END_VAR
_bResult := FALSE;

// Recover from premature stop
bGetPowerStatusBusy := TRUE;
_inst_intStep := intGetPowerStatusStep;

// Steps
(* TEMPLATE: Parameters should be added in step 10, and output
	parsing should be added in step 30. *)
CASE _inst_intStep OF
	0: // Wait for no error and router not busy
		IF NOT THIS^.P_bError AND NOT bRouterBusy THEN
			bRouterBusy := TRUE;
			_inst_intStep := _inst_intStep + 10;
		END_IF
		
	10: // Initialize parameters
		THIS^.M_LogMessage(_strSTART_MSG);
		_inst_fbParams.M_ClearParameters();
		_pArgs := _inst_fbParams.M_AddEmptyStruct('args');
		// TEMPLATE: Add any parameters here
		_inst_fbParams.M_OutputToParameterList(_inst_arrParams);
		_inst_intStep := _inst_intStep + 10;
		
	20: // Route the command
		_bComplete := M_RouterHelper(
			_in_strMethodName := _strCOMMAND_NAME, 
			_in_timeTimeout := _timeCOMMAND_TIMEOUT,
			_inout_arrParams := _inst_arrParams,
			_inout_arrOutputs := _inst_arrOutputs,
			_out_strReturnValue=>_inst_strRet);
		
		// If route completed, move to next step
		IF _bComplete THEN
			_inst_intStep := _inst_intStep + 10;
			bRouterBusy := FALSE;
		ELSIF THIS^.P_bError THEN
			_inst_intStep := 0;
			bRouterBusy := FALSE;
		END_IF
		
	30: // Parse results
		_intRet := STRING_TO_INT(_inst_strRet);
		IF _intRet > 0 THEN
			_bResult := TRUE;
			THIS^.M_LogMessage(_strEND_MSG);
			_inst_fbParams.M_LoadFromParameterList(_inst_arrOutputs);
			// TEMPLATE: Do any parsing here
			THIS^.bPoweredOn := _inst_fbParams.M_ParseBool(
				_inst_fbParams.M_GetParameter('poweredOn'));
			bPoweredOn := THIS^.bPoweredOn;
			
		// Set error if command failed
		ELSE
			THIS^.M_SetError(_udintERROR_ID, _strERROR_MSG);
		END_IF
		
		// Go back to start
		_inst_intStep := 0;
END_CASE

M_GetPowerStatus := _bResult;
intGetPowerStatusStep := _inst_intStep;
END_METHOD

(* This method should de-energize the device and then return TRUE once
	successful. P_bPoweredOn should be set to FALSE immediately when this is
	called unless the device is explicitly known to still be powered on. *)
METHOD M_PowerOff : BOOL
VAR CONSTANT
	_strCOMMAND_NAME : T_MaxString	:= 'PowerOff'; // Name of the API method
	_timeCOMMAND_TIMEOUT : TIME		:= T#30S; // Max time to receive API response
	_strSTART_MSG : T_MaxString		:= 'Powering off'; // Prints when method starts
	_strEND_MSG : T_MaxString		:= 'Powered off'; // Prints when method finishes
	_udintERROR_ID : UDINT			:= E_ApiDeviceError.FailedToPowerOff; // Error ID to set if command fails
	_strERROR_MSG : T_MaxString		:= 'Failed to power off!'; // Error message to set if command fails
END_VAR
VAR_INST
	_inst_arrParams: T_ApiParameterList; // Parameters array
	_inst_arrOutputs: T_ApiParameterList; // Outputs array
	_inst_strRet: T_ApiParamValue; // Return string from the router
	_inst_intStep: INT; // Current method step
	_inst_fbParams: FB_ApiParamBuilder; // Parameter builder FB
END_VAR
VAR
	_bComplete: BOOL; // True if the routing finishes
	_intRet: INT; // Return string converted to an integer
	_bResult : BOOL; // Output of the method
	_pArgs: PVOID; // Arguments pointer
END_VAR
_bResult := FALSE;

// Recover from premature stop
bPowerOffBusy := TRUE;
_inst_intStep := intPowerOffStep;

// Steps
(* TEMPLATE: Parameters should be added in step 10, and output
	parsing should be added in step 30. *)
CASE _inst_intStep OF
	0: // Wait for no error and router not busy
		IF NOT THIS^.P_bError AND NOT bRouterBusy THEN
			bRouterBusy := TRUE;
			_inst_intStep := _inst_intStep + 10;
		END_IF
		
	10: // Initialize parameters
		THIS^.M_LogMessage(_strSTART_MSG);
		_inst_fbParams.M_ClearParameters();
		_pArgs := _inst_fbParams.M_AddEmptyStruct('args');
		// TEMPLATE: Add any parameters here
		_inst_fbParams.M_OutputToParameterList(_inst_arrParams);
		_inst_intStep := _inst_intStep + 10;
		
	20: // Route the command
		_bComplete := M_RouterHelper(
			_in_strMethodName := _strCOMMAND_NAME, 
			_in_timeTimeout := _timeCOMMAND_TIMEOUT,
			_inout_arrParams := _inst_arrParams,
			_inout_arrOutputs := _inst_arrOutputs,
			_out_strReturnValue=>_inst_strRet);
		
		// If route completed, move to next step
		IF _bComplete THEN
			_inst_intStep := _inst_intStep + 10;
			bRouterBusy := FALSE;
		ELSIF THIS^.P_bError THEN
			_inst_intStep := 0;
			bRouterBusy := FALSE;
		END_IF
		
	30: // Parse results
		_intRet := STRING_TO_INT(_inst_strRet);
		IF _intRet > 0 THEN
			_bResult := TRUE;
			THIS^.M_LogMessage(_strEND_MSG);
			_inst_fbParams.M_LoadFromParameterList(_inst_arrOutputs);
			// TEMPLATE: Do any parsing here
			bPoweredOn := FALSE;
			
		// Set error if command failed
		ELSE
			THIS^.M_SetError(_udintERROR_ID, _strERROR_MSG);
		END_IF
		
		// Go back to start
		_inst_intStep := 0;
END_CASE

M_PowerOff := _bResult;
intPowerOffStep := _inst_intStep;
END_METHOD

(* This method should energize the device and then return TRUE and set
	P_bPoweredOn to TRUE once successful. *)
METHOD M_PowerOn : BOOL
VAR CONSTANT
	_strCOMMAND_NAME : T_MaxString	:= 'PowerOn'; // Name of the API method
	_timeCOMMAND_TIMEOUT : TIME		:= T#30S; // Max time to receive API response
	_strSTART_MSG : T_MaxString		:= 'Powering on'; // Prints when method starts
	_strEND_MSG : T_MaxString		:= 'Powered on'; // Prints when method finishes
	_udintERROR_ID : UDINT			:= E_ApiDeviceError.FailedToPowerOn; // Error ID to set if command fails
	_strERROR_MSG : T_MaxString		:= 'Failed to power on!'; // Error message to set if command fails
END_VAR
VAR_INST
	_inst_arrParams: T_ApiParameterList; // Parameters array
	_inst_arrOutputs: T_ApiParameterList; // Outputs array
	_inst_strRet: T_ApiParamValue; // Return string from the router
	_inst_intStep: INT; // Current method step
	_inst_fbParams: FB_ApiParamBuilder; // Parameter builder FB
END_VAR
VAR
	_bComplete: BOOL; // True if the routing finishes
	_intRet: INT; // Return string converted to an integer
	_bResult : BOOL; // Output of the method
	_pArgs: PVOID; // Arguments pointer
END_VAR
_bResult := FALSE;

// Recover from premature stop
bPowerOnBusy := TRUE;
_inst_intStep := intPowerOnStep;

// Steps
(* TEMPLATE: Parameters should be added in step 10, and output
	parsing should be added in step 30. *)
CASE _inst_intStep OF
	0: // Wait for no error and router not busy
		IF NOT THIS^.P_bError AND NOT bRouterBusy THEN
			bRouterBusy := TRUE;
			_inst_intStep := _inst_intStep + 10;
		END_IF
		
	10: // Initialize parameters
		THIS^.M_LogMessage(_strSTART_MSG);
		_inst_fbParams.M_ClearParameters();
		_pArgs := _inst_fbParams.M_AddEmptyStruct('args');
		// TEMPLATE: Add any parameters here
		_inst_fbParams.M_OutputToParameterList(_inst_arrParams);
		_inst_intStep := _inst_intStep + 10;
		
	20: // Route the command
		_bComplete := M_RouterHelper(
			_in_strMethodName := _strCOMMAND_NAME, 
			_in_timeTimeout := _timeCOMMAND_TIMEOUT,
			_inout_arrParams := _inst_arrParams,
			_inout_arrOutputs := _inst_arrOutputs,
			_out_strReturnValue=>_inst_strRet);
		
		// If route completed, move to next step
		IF _bComplete THEN
			_inst_intStep := _inst_intStep + 10;
			bRouterBusy := FALSE;
		ELSIF THIS^.P_bError THEN
			_inst_intStep := 0;
			bRouterBusy := FALSE;
		END_IF
		
	30: // Parse results
		_intRet := STRING_TO_INT(_inst_strRet);
		IF _intRet > 0 THEN
			_bResult := TRUE;
			THIS^.M_LogMessage(_strEND_MSG);
			_inst_fbParams.M_LoadFromParameterList(_inst_arrOutputs);
			// TEMPLATE: Do any parsing here
			bPoweredOn := TRUE;
			
		// Set error if command failed
		ELSE
			THIS^.M_SetError(_udintERROR_ID, _strERROR_MSG);
		END_IF
		
		// Go back to start
		_inst_intStep := 0;
END_CASE

M_PowerOn := _bResult;
intPowerOnStep := _inst_intStep;
END_METHOD

(* This property should be TRUE while any method in this interface is actively
	executing, or FALSE otherwise. *)
PROPERTY P_bPowerBusy : BOOL
GET
P_bPowerBusy := bRouterBusy;
END_GET
END_PROPERTY

(* This should be set to TRUE if M_PowerOn is successful or if M_GetPowerStatus
	determines that the device is powered on. Otherwise, this should be FALSE. *)
PROPERTY P_bPoweredOn : BOOL
GET
P_bPoweredOn := bPoweredOn;
END_GET
END_PROPERTY

(* This method should explicitly get the current program loaded on the device.
	If the current program is successfully gotten, this method should return
	TRUE and set P_strCurrentProgram and strCurrentProgram to the gotten
	program name. If this method fails, both should be set to empty strings. *)
METHOD M_GetCurrentProgram : BOOL
VAR_OUTPUT
	(* This should be set to the name of the currently loaded program if
		the method was successful, or a blank string otherwise. *)
	strCurrentProgram	: Sensata_Common.T_MaxString;
END_VAR
VAR CONSTANT
	_strCOMMAND_NAME : T_MaxString	:= 'GetCurrentProgram'; // Name of the API method
	_timeCOMMAND_TIMEOUT : TIME		:= T#10S; // Max time to receive API response
	_strSTART_MSG : T_MaxString		:= 'Getting current program'; // Prints when method starts
	_strEND_MSG : T_MaxString		:= 'Received current program'; // Prints when method finishes
	_udintERROR_ID : UDINT			:= E_ApiDeviceError.FailedToGetCurrentProgram; // Error ID to set if command fails
	_strERROR_MSG : T_MaxString		:= 'Failed to get current program!'; // Error message to set if command fails
END_VAR
VAR_INST
	_inst_arrParams: T_ApiParameterList; // Parameters array
	_inst_arrOutputs: T_ApiParameterList; // Outputs array
	_inst_strRet: T_ApiParamValue; // Return string from the router
	_inst_intStep: INT; // Current method step
	_inst_fbParams: FB_ApiParamBuilder; // Parameter builder FB
END_VAR
VAR
	_bComplete: BOOL; // True if the routing finishes
	_intRet: INT; // Return string converted to an integer
	_bResult : BOOL; // Output of the method
	_pArgs: PVOID; // Arguments pointer
END_VAR
_bResult := FALSE;

// Recover from premature stop
bGetCurrentProgramBusy := TRUE;
_inst_intStep := intGetCurrentProgramStep;

// Steps
(* TEMPLATE: Parameters should be added in step 10, and output
	parsing should be added in step 30. *)
CASE _inst_intStep OF
	0: // Wait for no error and router not busy
		IF NOT THIS^.P_bError AND NOT bRouterBusy THEN
			bRouterBusy := TRUE;
			_inst_intStep := _inst_intStep + 10;
		END_IF
		
	10: // Initialize parameters
		THIS^.M_LogMessage(_strSTART_MSG);
		_inst_fbParams.M_ClearParameters();
		_pArgs := _inst_fbParams.M_AddEmptyStruct('args');
		// TEMPLATE: Add any parameters here
		_inst_fbParams.M_OutputToParameterList(_inst_arrParams);
		_inst_intStep := _inst_intStep + 10;
		
	20: // Route the command
		_bComplete := M_RouterHelper(
			_in_strMethodName := _strCOMMAND_NAME, 
			_in_timeTimeout := _timeCOMMAND_TIMEOUT,
			_inout_arrParams := _inst_arrParams,
			_inout_arrOutputs := _inst_arrOutputs,
			_out_strReturnValue=>_inst_strRet);
		
		// If route completed, move to next step
		IF _bComplete THEN
			_inst_intStep := _inst_intStep + 10;
			bRouterBusy := FALSE;
		ELSIF THIS^.P_bError THEN
			_inst_intStep := 0;
			bRouterBusy := FALSE;
		END_IF
		
	30: // Parse results
		_intRet := STRING_TO_INT(_inst_strRet);
		IF _intRet > 0 THEN
			_bResult := TRUE;
			THIS^.M_LogMessage(_strEND_MSG);
			_inst_fbParams.M_LoadFromParameterList(_inst_arrOutputs);
			// TEMPLATE: Do any parsing here
			THIS^.strLoadedProgram := _inst_fbParams.M_ParseString(
				_inst_fbParams.M_GetParameter('programName'));
			strCurrentProgram := THIS^.strLoadedProgram;
			
		// Set error if command failed
		ELSE
			THIS^.M_SetError(_udintERROR_ID, _strERROR_MSG);
		END_IF
		
		// Go back to start
		_inst_intStep := 0;
END_CASE

M_GetCurrentProgram := _bResult;
intGetCurrentProgramStep := _inst_intStep;
END_METHOD

(* This method should explicitly check the program state of the device.
	Once the program state is known, this method should return TRUE and set
	P_enumProgramState and enumProgramState to the relevant E_ProgramState
	value, else it should set both to E_ProgramState.Unknown. *)
METHOD M_GetProgramState : BOOL
VAR_OUTPUT
	(* If the program state is successfully gotten, this should be set to
		the relevant E_ProgramState value. If this method fails, this should
		be set to E_ProgramState.Unknown. *)
	enumProgramState	: Sensata_Common.E_ProgramState;
END_VAR
VAR CONSTANT
	_strCOMMAND_NAME : T_MaxString	:= 'GetControlState'; // Name of the API method
	_timeCOMMAND_TIMEOUT : TIME		:= T#10S; // Max time to receive API response
	_strSTART_MSG : T_MaxString		:= 'Getting program state'; // Prints when method starts
	_strEND_MSG : T_MaxString		:= 'Received program state'; // Prints when method finishes
	_udintERROR_ID : UDINT			:= E_ApiDeviceError.FailedToGetProgramState; // Error ID to set if command fails
	_strERROR_MSG : T_MaxString		:= 'Failed to get program state!'; // Error message to set if command fails
END_VAR
VAR_INST
	_inst_arrParams: T_ApiParameterList; // Parameters array
	_inst_arrOutputs: T_ApiParameterList; // Outputs array
	_inst_strRet: T_ApiParamValue; // Return string from the router
	_inst_intStep: INT; // Current method step
	_inst_fbParams: FB_ApiParamBuilder; // Parameter builder FB
END_VAR
VAR
	_bComplete: BOOL; // True if the routing finishes
	_intRet: INT; // Return string converted to an integer
	_bResult : BOOL; // Output of the method
	_pArgs: PVOID; // Arguments pointer
	dintControlState: DINT; // Current program state
END_VAR
_bResult := FALSE;

// Recover from premature stop
bGetProgramStateBusy := TRUE;
_inst_intStep := intGetProgramStateStep;

// Steps
(* TEMPLATE: Parameters should be added in step 10, and output
	parsing should be added in step 30. *)
CASE _inst_intStep OF
	0: // Wait for no error and router not busy
		IF NOT THIS^.P_bError AND NOT bRouterBusy THEN
			bRouterBusy := TRUE;
			_inst_intStep := _inst_intStep + 10;
		END_IF
		
	10: // Initialize parameters
		THIS^.M_LogMessage(_strSTART_MSG);
		_inst_fbParams.M_ClearParameters();
		_pArgs := _inst_fbParams.M_AddEmptyStruct('args');
		// TEMPLATE: Add any parameters here
		_inst_fbParams.M_OutputToParameterList(_inst_arrParams);
		_inst_intStep := _inst_intStep + 10;
		
	20: // Route the command
		_bComplete := M_RouterHelper(
			_in_strMethodName := _strCOMMAND_NAME, 
			_in_timeTimeout := _timeCOMMAND_TIMEOUT,
			_inout_arrParams := _inst_arrParams,
			_inout_arrOutputs := _inst_arrOutputs,
			_out_strReturnValue=>_inst_strRet);
		
		// If route completed, move to next step
		IF _bComplete THEN
			_inst_intStep := _inst_intStep + 10;
			bRouterBusy := FALSE;
		ELSIF THIS^.P_bError THEN
			_inst_intStep := 0;
			bRouterBusy := FALSE;
		END_IF
		
	30: // Parse results
		_intRet := STRING_TO_INT(_inst_strRet);
		IF _intRet > 0 THEN
			_bResult := TRUE;
			THIS^.M_LogMessage(_strEND_MSG);
			_inst_fbParams.M_LoadFromParameterList(_inst_arrOutputs);
			// TEMPLATE: Do any parsing here
			dintControlState := _inst_fbParams.M_ParseInt(_inst_fbParams.M_GetParameter('state'));
			CASE dintControlState OF
				0: enumProgramState := E_ProgramState.Unknown;
				1: enumProgramState := E_ProgramState.Stopped;
				2: enumProgramState := E_ProgramState.Running;
				3: enumProgramState := E_ProgramState.Paused;
			ELSE
				enumProgramState := E_ProgramState.Unknown;
			END_CASE
			THIS^.enumProgramState := enumProgramState;
			
		// Set error if command failed
		ELSE
			THIS^.M_SetError(_udintERROR_ID, _strERROR_MSG);
		END_IF
		
		// Go back to start
		_inst_intStep := 0;
END_CASE

M_GetProgramState := _bResult;
intGetProgramStateStep := _inst_intStep;
END_METHOD

(* This method should load a new program onto the device, and then return TRUE
	once program loading is completed. Once this method begins the program loading
	process, P_strCurrentProgram should be cleared unless it is still explicitly
	known to be loaded. *)
METHOD M_LoadProgram : BOOL
VAR_INPUT
END_VAR
VAR CONSTANT
	_strCOMMAND_NAME : T_MaxString	:= 'LoadProgram'; // Name of the API method
	_timeCOMMAND_TIMEOUT : TIME		:= T#30S; // Max time to receive API response
	_strSTART_MSG : T_MaxString		:= 'Loading program'; // Prints when method starts
	_strEND_MSG : T_MaxString		:= 'Loaded program'; // Prints when method finishes
	_udintERROR_ID : UDINT			:= E_ApiDeviceError.FailedToLoadProgram; // Error ID to set if command fails
	_strERROR_MSG : T_MaxString		:= 'Failed to load program!'; // Error message to set if command fails
END_VAR
VAR_INST
	_inst_arrParams: T_ApiParameterList; // Parameters array
	_inst_arrOutputs: T_ApiParameterList; // Outputs array
	_inst_strRet: T_ApiParamValue; // Return string from the router
	_inst_intStep: INT; // Current method step
	_inst_fbParams: FB_ApiParamBuilder; // Parameter builder FB
END_VAR
VAR
	_bComplete: BOOL; // True if the routing finishes
	_intRet: INT; // Return string converted to an integer
	_bResult : BOOL; // Output of the method
	_pArgs: PVOID; // Arguments pointer
END_VAR
_bResult := FALSE;

// Recover from premature stop
bLoadProgramBusy := TRUE;
_inst_intStep := intLoadProgramStep;

// Steps
(* TEMPLATE: Parameters should be added in step 10, and output
	parsing should be added in step 30. *)
CASE _inst_intStep OF
	0: // Wait for no error and router not busy
		IF NOT THIS^.P_bError AND NOT bRouterBusy THEN
			bRouterBusy := TRUE;
			_inst_intStep := _inst_intStep + 10;
		END_IF
		
	10: // Initialize parameters
		THIS^.M_LogMessage(_strSTART_MSG);
		_inst_fbParams.M_ClearParameters();
		_pArgs := _inst_fbParams.M_AddEmptyStruct('args');
		_inst_fbParams.M_AddStructMember(_pArgs,'programNumber', in_intProgramNum);
		_inst_fbParams.M_AddStructMember(_pArgs,'Mode', in_intWobbleMode);
		_inst_fbParams.M_AddStructMember(_pArgs,'Frequency', in_intWobbleFreq);
		_inst_fbParams.M_AddStructMember(_pArgs,'Amplitude', in_lrWobbleAmp);
		_inst_fbParams.M_AddStructMember(_pArgs,'offset', in_intWobbleOffset);
		_inst_fbParams.M_AddStructMember(_pArgs,'MaterialSpeed', in_intMaterialSpeed);
		_inst_fbParams.M_AddStructMember(_pArgs,'Save', in_intSaveSetting);
		//_inst_fbParams.M_AddStructMember(_pArgs, 'programName', '');
		_inst_fbParams.M_OutputToParameterList(_inst_arrParams);
		_inst_intStep := _inst_intStep + 10;
		
	20: // Route the command
		_bComplete := M_RouterHelper(
			_in_strMethodName := _strCOMMAND_NAME, 
			_in_timeTimeout := _timeCOMMAND_TIMEOUT,
			_inout_arrParams := _inst_arrParams,
			_inout_arrOutputs := _inst_arrOutputs,
			_out_strReturnValue=>_inst_strRet);
		
		// If route completed, move to next step
		IF _bComplete THEN
			_inst_intStep := _inst_intStep + 10;
			bRouterBusy := FALSE;
		ELSIF THIS^.P_bError THEN
			_inst_intStep := 0;
			bRouterBusy := FALSE;
		END_IF
		
	30: // Parse results
		_intRet := STRING_TO_INT(_inst_strRet);
		IF _intRet > 0 THEN
			_bResult := TRUE;
			THIS^.M_LogMessage(_strEND_MSG);
			_inst_fbParams.M_LoadFromParameterList(_inst_arrOutputs);
			// TEMPLATE: Do any parsing here
			strLoadedProgram := '';
			
		// Set error if command failed
		ELSE
			THIS^.M_SetError(_udintERROR_ID, _strERROR_MSG);
		END_IF
		
		// Go back to start
		_inst_intStep := 0;
END_CASE

M_LoadProgram := _bResult;
intLoadProgramStep := _inst_intStep;
END_METHOD

(* This program should move to the program state from whatever state it was in
	to the Paused state, and then return TRUE once successful. If the program
	state is Stopped, this method should return TRUE but keep the current state
	as Stopped, since Paused at the beginning at the program is equivalent to
	being Stopped. *)
METHOD M_PauseProgram : BOOL
VAR CONSTANT
	_strCOMMAND_NAME : T_MaxString	:= 'PauseProgram'; // Name of the API method
	_timeCOMMAND_TIMEOUT : TIME		:= T#30S; // Max time to receive API response
	_strSTART_MSG : T_MaxString		:= 'Pausing program'; // Prints when method starts
	_strEND_MSG : T_MaxString		:= 'Paused program'; // Prints when method finishes
	_udintERROR_ID : UDINT			:= E_ApiDeviceError.FailedToPauseProgram; // Error ID to set if command fails
	_strERROR_MSG : T_MaxString		:= 'Failed to pause program!'; // Error message to set if command fails
END_VAR
VAR_INST
	_inst_arrParams: T_ApiParameterList; // Parameters array
	_inst_arrOutputs: T_ApiParameterList; // Outputs array
	_inst_strRet: T_ApiParamValue; // Return string from the router
	_inst_intStep: INT; // Current method step
	_inst_fbParams: FB_ApiParamBuilder; // Parameter builder FB
END_VAR
VAR
	_bComplete: BOOL; // True if the routing finishes
	_intRet: INT; // Return string converted to an integer
	_bResult : BOOL; // Output of the method
	_pArgs: PVOID; // Arguments pointer
END_VAR
_bResult := FALSE;

// Recover from premature stop
bPauseProgramBusy := TRUE;
_inst_intStep := intPauseProgramStep;

// Steps
(* TEMPLATE: Parameters should be added in step 10, and output
	parsing should be added in step 30. *)
CASE _inst_intStep OF
	0: // Wait for no error and router not busy
		IF NOT THIS^.P_bError AND NOT bRouterBusy THEN
			bRouterBusy := TRUE;
			_inst_intStep := _inst_intStep + 10;
		END_IF
		
	10: // Initialize parameters
		THIS^.M_LogMessage(_strSTART_MSG);
		_inst_fbParams.M_ClearParameters();
		_pArgs := _inst_fbParams.M_AddEmptyStruct('args');
		// TEMPLATE: Add any parameters here
		_inst_fbParams.M_OutputToParameterList(_inst_arrParams);
		_inst_intStep := _inst_intStep + 10;
		
	20: // Route the command
		_bComplete := M_RouterHelper(
			_in_strMethodName := _strCOMMAND_NAME, 
			_in_timeTimeout := _timeCOMMAND_TIMEOUT,
			_inout_arrParams := _inst_arrParams,
			_inout_arrOutputs := _inst_arrOutputs,
			_out_strReturnValue=>_inst_strRet);
		
		// If route completed, move to next step
		IF _bComplete THEN
			_inst_intStep := _inst_intStep + 10;
			bRouterBusy := FALSE;
		ELSIF THIS^.P_bError THEN
			_inst_intStep := 0;
			bRouterBusy := FALSE;
		END_IF
		
	30: // Parse results
		_intRet := STRING_TO_INT(_inst_strRet);
		IF _intRet > 0 THEN
			_bResult := TRUE;
			THIS^.M_LogMessage(_strEND_MSG);
			_inst_fbParams.M_LoadFromParameterList(_inst_arrOutputs);
			// TEMPLATE: Do any parsing here
			enumProgramState := E_ProgramState.Paused;
			
		// Set error if command failed
		ELSE
			THIS^.M_SetError(_udintERROR_ID, _strERROR_MSG);
		END_IF
		
		// Go back to start
		_inst_intStep := 0;
END_CASE

M_PauseProgram := _bResult;
intPauseProgramStep := _inst_intStep;
END_METHOD

(* This should move the program state from whatever state it is in to the
	Running state, and then return TRUE once successful. Starting from the
	Paused state should always continue execution from whatever point the
	program was at when the program was initially paused. *)
METHOD M_StartProgram : BOOL
VAR CONSTANT
	_strCOMMAND_NAME : T_MaxString	:= 'StartProgram'; // Name of the API method
	_timeCOMMAND_TIMEOUT : TIME		:= T#30S; // Max time to receive API response
	_strSTART_MSG : T_MaxString		:= 'Starting program'; // Prints when method starts
	_strEND_MSG : T_MaxString		:= 'Started program'; // Prints when method finishes
	_udintERROR_ID : UDINT			:= E_ApiDeviceError.FailedToStartProgram; // Error ID to set if command fails
	_strERROR_MSG : T_MaxString		:= 'Failed to start program!'; // Error message to set if command fails
END_VAR
VAR_INST
	_inst_arrParams: T_ApiParameterList; // Parameters array
	_inst_arrOutputs: T_ApiParameterList; // Outputs array
	_inst_strRet: T_ApiParamValue; // Return string from the router
	_inst_intStep: INT; // Current method step
	_inst_fbParams: FB_ApiParamBuilder; // Parameter builder FB
END_VAR
VAR
	_bComplete: BOOL; // True if the routing finishes
	_intRet: INT; // Return string converted to an integer
	_bResult : BOOL; // Output of the method
	_pArgs: PVOID; // Arguments pointer
END_VAR
_bResult := FALSE;

// Recover from premature stop
bStartProgramBusy := TRUE;
_inst_intStep := intStartProgramStep;

// Steps
(* TEMPLATE: Parameters should be added in step 10, and output
	parsing should be added in step 30. *)
CASE _inst_intStep OF
	0: // Wait for no error and router not busy
		IF NOT THIS^.P_bError AND NOT bRouterBusy THEN
			bRouterBusy := TRUE;
			_inst_intStep := _inst_intStep + 10;
		END_IF
		
	10: // Initialize parameters
		THIS^.M_LogMessage(_strSTART_MSG);
		_inst_fbParams.M_ClearParameters();
		_pArgs := _inst_fbParams.M_AddEmptyStruct('args');
		// TEMPLATE: Add any parameters here
		_inst_fbParams.M_OutputToParameterList(_inst_arrParams);
		_inst_intStep := _inst_intStep + 10;
		
	20: // Route the command
		_bComplete := M_RouterHelper(
			_in_strMethodName := _strCOMMAND_NAME, 
			_in_timeTimeout := _timeCOMMAND_TIMEOUT,
			_inout_arrParams := _inst_arrParams,
			_inout_arrOutputs := _inst_arrOutputs,
			_out_strReturnValue=>_inst_strRet);
		
		// If route completed, move to next step
		IF _bComplete THEN
			_inst_intStep := _inst_intStep + 10;
			bRouterBusy := FALSE;
		ELSIF THIS^.P_bError THEN
			_inst_intStep := 0;
			bRouterBusy := FALSE;
		END_IF
		
	30: // Parse results
		_intRet := STRING_TO_INT(_inst_strRet);
		IF _intRet > 0 THEN
			_bResult := TRUE;
			THIS^.M_LogMessage(_strEND_MSG);
			_inst_fbParams.M_LoadFromParameterList(_inst_arrOutputs);
			// TEMPLATE: Do any parsing here
			enumProgramState := E_ProgramState.Running;
			
		// Set error if command failed
		ELSE
			THIS^.M_SetError(_udintERROR_ID, _strERROR_MSG);
		END_IF
		
		// Go back to start
		_inst_intStep := 0;
END_CASE

M_StartProgram := _bResult;
intStartProgramStep := _inst_intStep;
END_METHOD

(* This should change the program state from whatever state it was in to the
	Stopped state and then return TRUE. Moving to the Stopped state should
	always reset the program execution back to the beginning. *)
METHOD M_StopProgram : BOOL
VAR CONSTANT
	_strCOMMAND_NAME : T_MaxString	:= 'StopProgram'; // Name of the API method
	_timeCOMMAND_TIMEOUT : TIME		:= T#30S; // Max time to receive API response
	_strSTART_MSG : T_MaxString		:= 'Stopping'; // Prints when method starts
	_strEND_MSG : T_MaxString		:= 'Stopped'; // Prints when method finishes
	_udintERROR_ID : UDINT			:= E_ApiDeviceError.FailedToStopProgram; // Error ID to set if command fails
	_strERROR_MSG : T_MaxString		:= 'Failed to stop program!'; // Error message to set if command fails
END_VAR
VAR_INST
	_inst_arrParams: T_ApiParameterList; // Parameters array
	_inst_arrOutputs: T_ApiParameterList; // Outputs array
	_inst_strRet: T_ApiParamValue; // Return string from the router
	_inst_intStep: INT; // Current method step
	_inst_fbParams: FB_ApiParamBuilder; // Parameter builder FB
END_VAR
VAR
	_bComplete: BOOL; // True if the routing finishes
	_intRet: INT; // Return string converted to an integer
	_bResult : BOOL; // Output of the method
	_pArgs: PVOID; // Arguments pointer
END_VAR
_bResult := FALSE;

// Recover from premature stop
bStopProgramBusy := TRUE;
_inst_intStep := intStopProgramStep;

// Steps
(* TEMPLATE: Parameters should be added in step 10, and output
	parsing should be added in step 30. *)
CASE _inst_intStep OF
	0: // Wait for no error and router not busy
		IF NOT THIS^.P_bError AND NOT bRouterBusy THEN
			bRouterBusy := TRUE;
			_inst_intStep := _inst_intStep + 10;
		END_IF
		
	10: // Initialize parameters
		THIS^.M_LogMessage(_strSTART_MSG);
		_inst_fbParams.M_ClearParameters();
		_pArgs := _inst_fbParams.M_AddEmptyStruct('args');
		// TEMPLATE: Add any parameters here
		_inst_fbParams.M_OutputToParameterList(_inst_arrParams);
		_inst_intStep := _inst_intStep + 10;
		
	20: // Route the command
		_bComplete := M_RouterHelper(
			_in_strMethodName := _strCOMMAND_NAME, 
			_in_timeTimeout := _timeCOMMAND_TIMEOUT,
			_inout_arrParams := _inst_arrParams,
			_inout_arrOutputs := _inst_arrOutputs,
			_out_strReturnValue=>_inst_strRet);
		
		// If route completed, move to next step
		IF _bComplete THEN
			_inst_intStep := _inst_intStep + 10;
			bRouterBusy := FALSE;
		ELSIF THIS^.P_bError THEN
			_inst_intStep := 0;
			bRouterBusy := FALSE;
		END_IF
		
	30: // Parse results
		_intRet := STRING_TO_INT(_inst_strRet);
		IF _intRet > 0 THEN
			_bResult := TRUE;
			THIS^.M_LogMessage(_strEND_MSG);
			_inst_fbParams.M_LoadFromParameterList(_inst_arrOutputs);
			// TEMPLATE: Do any parsing here
			enumProgramState := E_ProgramState.Stopped;
			
		// Set error if command failed
		ELSE
			THIS^.M_SetError(_udintERROR_ID, _strERROR_MSG);
		END_IF
		
		// Go back to start
		_inst_intStep := 0;
END_CASE

M_StopProgram := _bResult;
intStopProgramStep := _inst_intStep;
END_METHOD

(* This property should be TRUE while any method in this interface is actively
	executing, or FALSE otherwise. *)
PROPERTY P_bProgramControlBusy : BOOL
GET
P_bProgramControlBusy := bRouterBusy;
END_GET
END_PROPERTY

(* The current E_ProgramState value of the device. This should be reset to
	E_ProgramState.Unknown if any methods in this interface interact with the
	device but fail. *)
PROPERTY P_enumProgramState : Sensata_Common.E_ProgramState
GET
P_enumProgramState := enumProgramState;
END_GET
END_PROPERTY

(* The value of the currently loaded program. This should only be set by
	M_LoadProgram or M_GetCurrentProgram, and set to a blank string if either
	fail. *)
PROPERTY P_strCurrentProgram : Sensata_Common.T_MaxString
GET
P_strCurrentProgram := strLoadedProgram;
END_GET
END_PROPERTY

(* This method should establish any external connections required to use the
	functions of the device, and return TRUE and set P_bConnected to TRUE once
	connected. *)
METHOD M_Reset : BOOL
VAR CONSTANT
	_strCOMMAND_NAME : T_MaxString	:= 'Reset'; // Name of the API method
	_timeCOMMAND_TIMEOUT : TIME		:= T#30S; // Max time to receive API response
	_strSTART_MSG : T_MaxString		:= 'Resetting'; // Prints when method starts
	_strEND_MSG : T_MaxString		:= 'Reset'; // Prints when method finishes
	_udintERROR_ID : UDINT			:= E_ApiDeviceError.FailedToReset; // Error ID to set if command fails
	_strERROR_MSG : T_MaxString		:= 'Failed to reset!'; // Error message to set if command fails
END_VAR
VAR_INST
	_inst_arrParams: T_ApiParameterList; // Parameters array
	_inst_arrOutputs: T_ApiParameterList; // Outputs array
	_inst_strRet: T_ApiParamValue; // Return string from the router
	_inst_intStep: INT; // Current method step
	_inst_fbParams: FB_ApiParamBuilder; // Parameter builder FB
END_VAR
VAR
	_bComplete: BOOL; // True if the routing finishes
	_intRet: INT; // Return string converted to an integer
	_bResult : BOOL; // Output of the method
	_pArgs: PVOID; // Arguments pointer
END_VAR
_bResult := FALSE;

// Recover from premature stop
bResetBusy := TRUE;
_inst_intStep := intResetStep;

// Steps
(* TEMPLATE: Parameters should be added in step 10, and output
	parsing should be added in step 30. *)
CASE _inst_intStep OF
	0: // Wait for no error and router not busy
		IF (NOT THIS^.P_bError) AND (NOT bRouterBusy) AND THIS^.P_bConnected THEN
			bRouterBusy := TRUE;
			_inst_intStep := _inst_intStep + 10;
		ELSIF (NOT THIS^.P_bError) AND (NOT THIS^.P_bConnected) THEN
			_bResult := TRUE;
		END_IF
		
	10: // Initialize parameters
		THIS^.M_LogMessage(_strSTART_MSG);
		_inst_fbParams.M_ClearParameters();
		_pArgs := _inst_fbParams.M_AddEmptyStruct('args');
		// TEMPLATE: Add any parameters here
		_inst_fbParams.M_OutputToParameterList(_inst_arrParams);
		_inst_intStep := _inst_intStep + 10;
		
	20: // Route the command
		_bComplete := M_RouterHelper(
			_in_strMethodName := _strCOMMAND_NAME, 
			_in_timeTimeout := _timeCOMMAND_TIMEOUT,
			_inout_arrParams := _inst_arrParams,
			_inout_arrOutputs := _inst_arrOutputs,
			_out_strReturnValue=>_inst_strRet);
		
		// If route completed, move to next step
		IF _bComplete THEN
			_inst_intStep := _inst_intStep + 10;
			bRouterBusy := FALSE;
		ELSIF THIS^.P_bError THEN
			_inst_intStep := 0;
			bRouterBusy := FALSE;
		END_IF
		
	30: // Parse results
		_intRet := STRING_TO_INT(_inst_strRet);
		IF _intRet >= 0 THEN
			_bResult := TRUE;
			THIS^.M_LogMessage(_strEND_MSG);
			_inst_fbParams.M_LoadFromParameterList(_inst_arrOutputs);
			// TEMPLATE: Do any parsing here
			bConnected := TRUE;
			
		// Set error if command failed
		ELSE
			THIS^.M_SetError(_udintERROR_ID, _strERROR_MSG);
		END_IF
		
		// Go back to start
		_inst_intStep := 0;
END_CASE

M_Reset := _bResult;
intResetStep := _inst_intStep;
END_METHOD

(* This property should be TRUE while any method in this interface is actively
	executing, or FALSE otherwise. *)
PROPERTY P_bResetBusy : BOOL
GET
P_bResetBusy := bResetBusy;
END_GET
END_PROPERTY

ACTION A_CommandRecovery:
(*
	Tell methods to reset if they were not called in the last cycle.
	Make sure to call A_CommandRecovery in function block body.
*)



IF NOT bConnectBusy AND intConnectStep > 0 THEN
	intConnectStep := 0;
	bRouterBusy := FALSE;
	THIS^.M_LogWarning('M_Connect ended prematurely!');
END_IF
bConnectBusy := FALSE;

IF NOT bDisconnectBusy AND intDisconnectStep > 0 THEN
	intDisconnectStep := 0;
	bRouterBusy := FALSE;
	THIS^.M_LogWarning('M_Disconnect ended prematurely!');
END_IF
bDisconnectBusy := FALSE;

IF NOT bGetConnectStatusBusy AND intGetConnectStatusStep > 0 THEN
	intGetConnectStatusStep := 0;
	bRouterBusy := FALSE;
	THIS^.M_LogWarning('M_GetConnectStatus ended prematurely!');
END_IF
bGetConnectStatusBusy := FALSE;

IF NOT bEnableBusy AND intEnableStep > 0 THEN
	intEnableStep := 0;
	bRouterBusy := FALSE;
	THIS^.M_LogWarning('M_Enable ended prematurely!');
END_IF
bEnableBusy := FALSE;

IF NOT bDisableBusy AND intDisableStep > 0 THEN
	intDisableStep := 0;
	bRouterBusy := FALSE;
	THIS^.M_LogWarning('M_Disable ended prematurely!');
END_IF
bDisableBusy := FALSE;

IF NOT bGetEnableStatusBusy AND intGetEnableStatusStep > 0 THEN
	intGetEnableStatusStep := 0;
	bRouterBusy := FALSE;
	THIS^.M_LogWarning('M_GetEnableStatus ended prematurely!');
END_IF
bGetEnableStatusBusy := FALSE;

IF NOT bPowerOnBusy AND intPowerOnStep > 0 THEN
	intPowerOnStep := 0;
	bRouterBusy := FALSE;
	THIS^.M_LogWarning('M_PowerOn ended prematurely!');
END_IF
bPowerOnBusy := FALSE;

IF NOT bPowerOffBusy AND intPowerOffStep > 0 THEN
	intPowerOffStep := 0;
	bRouterBusy := FALSE;
	THIS^.M_LogWarning('M_PowerOff ended prematurely!');
END_IF
bPowerOffBusy := FALSE;

IF NOT bGetPowerStatusBusy AND intGetPowerStatusStep > 0 THEN
	intGetPowerStatusStep := 0;
	bRouterBusy := FALSE;
	THIS^.M_LogWarning('M_GetPowerStatus ended prematurely!');
END_IF
bGetPowerStatusBusy := FALSE;

IF NOT bGetCurrentProgramBusy AND intGetCurrentProgramStep > 0 THEN
	intGetCurrentProgramStep := 0;
	bRouterBusy := FALSE;
	THIS^.M_LogWarning('M_GetCurrentProgram ended prematurely!');
END_IF
bGetCurrentProgramBusy := FALSE;

IF NOT bGetProgramStateBusy AND intGetProgramStateStep > 0 THEN
	intGetProgramStateStep := 0;
	bRouterBusy := FALSE;
	THIS^.M_LogWarning('M_GetProgramState ended prematurely!');
END_IF
bGetProgramStateBusy := FALSE;

IF NOT bLoadProgramBusy AND intLoadProgramStep > 0 THEN
	intLoadProgramStep := 0;
	bRouterBusy := FALSE;
	THIS^.M_LogWarning('M_LoadProgram ended prematurely!');
END_IF
bLoadProgramBusy := FALSE;

IF NOT bPauseProgramBusy AND intPauseProgramStep > 0 THEN
	intPauseProgramStep := 0;
	bRouterBusy := FALSE;
	THIS^.M_LogWarning('M_PauseProgram ended prematurely!');
END_IF
bPauseProgramBusy := FALSE;

IF NOT bStartProgramBusy AND intStartProgramStep > 0 THEN
	intStartProgramStep := 0;
	bRouterBusy := FALSE;
	THIS^.M_LogWarning('M_StartProgram ended prematurely!');
END_IF
bStartProgramBusy := FALSE;

IF NOT bStopProgramBusy AND intStopProgramStep > 0 THEN
	intStopProgramStep := 0;
	bRouterBusy := FALSE;
	THIS^.M_LogWarning('M_StopProgram ended prematurely!');
END_IF
bStopProgramBusy := FALSE;

IF NOT bResetBusy AND intResetStep > 0 THEN
	intResetStep := 0;
	bRouterBusy := FALSE;
	THIS^.M_LogWarning('M_ResetBusy ended prematurely!');
END_IF
bResetBusy := FALSE;

IF NOT bAbortBusy AND intAbortStep > 0 THEN
	intAbortStep := 0;
	bRouterBusy := FALSE;
	THIS^.M_LogWarning('M_Abort ended prematurely!');
END_IF
bAbortBusy := FALSE;

IF NOT bRouterHelperBusy AND intRouterHelperStep > 0 THEN
	intRouterHelperStep := 0;
	bRouterBusy := FALSE;
	THIS^.M_LogWarning('M_RouterHelper ended prematurely!');
END_IF
bRouterHelperBusy := FALSE;
END_ACTION

(*
Sends the given method to the API and receives and partially parses the result.
*)
METHOD PRIVATE M_RouterHelper : BOOL
VAR_INPUT
	(* Name of the method to call. *)
	_in_strMethodName : T_MaxString;
	(* Maximum time to wait for method response. *)
	_in_timeTimeout : TIME;
END_VAR
VAR_IN_OUT
	(* The array of parameters to send to the API. *)
	_inout_arrParams : T_ApiParameterList;
	(* The array that gets populated with any method output data. *)
	_inout_arrOutputs : T_ApiParameterList;
END_VAR
VAR_OUTPUT
	(* JSON string of the method return value. *)
	_out_strReturnValue: T_ApiParamValue;
END_VAR
VAR_INST
	(* Current step. *)
	_inst_intStep: INT;
	(* True if the method executed. *)
	_inst_bExec: BOOL;
	(* Return string of the method. *)
	_inst_strRet: T_ApiParamValue;
END_VAR
VAR
	(* True once the command routing finishes. *)
	_bComplete: BOOL;
	(* True once the API connects. *)
	_bApiConnect: BOOL;
END_VAR
// Recover from premature stop
bRouterHelperBusy := TRUE;
_inst_intStep := intRouterHelperStep;

// Steps
CASE _inst_intStep OF
	0: // Start process only if there is no error on this FB
		IF NOT THIS^.P_bError THEN
			in_fbApi.M_ClearError();
			_inst_intStep := 10;
		END_IF
		
	10: // Check if command router is connected
		IF NOT in_fbApi.P_bConnected THEN
			_inst_intStep := 20; // Go to API connect step
		ELSE
			_inst_intStep := 30; // Go to route command step
		END_IF
		
	20: // Connect to the command router
		_bApiConnect := in_fbApi.M_Connect();
		IF _bApiConnect THEN
			_inst_intStep := _inst_intStep + 10; // Go to next step
		ELSIF in_fbApi.P_bError THEN
			THIS^.M_SetError(E_ApiDeviceError.CommandRouterError, 'Error on command router function block while connecting!');
			_inst_intStep := 0; // Go back to start
		END_IF
		
	30:	// Route the command
		_bComplete := in_fbApi.M_RouteCommand(
			_in_strModuleId := in_strApiModuleId,
			_in_strMethodName := _in_strMethodName,
			_in_timeTimeout := _in_timeTimeout,
			_inout_arrParameters := _inout_arrParams,
			_inout_arrOutputs := _inout_arrOutputs,
			_out_bCommandExecuted => _inst_bExec,
			_out_strReturnValue => _inst_strRet);
		IF _bComplete THEN
			_inst_intStep := _inst_intStep + 10; // Go to next step
		ELSIF in_fbApi.P_bError THEN
			THIS^.M_SetError(E_ApiDeviceError.CommandRouterError, 'Error on command router function block while routing command!');
			_inst_intStep := 0; // Go back to start
		END_IF
		
	40: // Check result then go back to start
		IF NOT _inst_bExec THEN
			THIS^.M_SetError(E_ApiDeviceError.CommandFault, 'Method in API failed to execute!');
		ELSE
			_out_strReturnValue := _inst_strRet;
			M_RouterHelper := TRUE;
		END_IF
		_inst_intStep := 0; // Go back to start
END_CASE

intRouterHelperStep := _inst_intStep;
END_METHOD

END_FUNCTION_BLOCK

// Concrete/IPG/FB_IPGWeld
(*
	Function block for controlling an IPG laser scanner from IPGWeld through
	the Modular API.

	First release: July 2023 Kevin Sanita <ksanita@sensata.com>
	
	Feb 2024: Renamed from FB_IPGLaser to FB_IPGWeld
*)
FUNCTION_BLOCK FB_IPGWeld EXTENDS FB_LaserScanner
	IMPLEMENTS 
		I_Abortable,
		I_Connectable, 
		I_Powerable,
		I_Enableable,
		I_Resettable,
		I_Programmable,
		I_Triggerable
VAR_INPUT
	(* Reference to an FB_CommandRouter function block to send commands
		to a command router in the API. *)
	in_fbApi : REFERENCE TO FB_CommandRouter;
	(* ID of the API module to send router commands to. *)
	in_strApiModuleId: T_MaxString;
	(* Name of the scanner in the IPGScan software. *)
	in_strScannerName: T_MaxString;
	(* Name of the program to load and trigger. *)
	in_strProgramName: T_MaxString;
	(* Enables the guide when triggering. *)
	in_bGuide: BOOL;
	(* Enables dry run mode when triggering. *)
	in_bDryrun: BOOL;
	(* Enables file saving while triggering. *)
	in_bSaveFile: BOOL;
	(* Explicitly disables the signal monitor while triggering. *)
	in_bSignalMonitorOff: BOOL;
	(* Explicitly enables the signal monitor while triggering. *)
	in_bSignalMonitorOn: BOOL;
	(* Runs the program subgroup with the given name. *)
	in_strGroup: T_MaxString;
END_VAR
VAR_IN_OUT
END_VAR
VAR_OUTPUT
END_VAR
VAR CONSTANT
END_VAR
VAR
	bConnected: BOOL; // Value of P_bConnected
	bEnabled: BOOL; // Value of P_bEnabled
	bPoweredOn: BOOL; // Value of P_bPoweredOn
	strLoadedProgram: STRING(255); // Value of P_strLoadedProgram
	enumProgramState: E_PROGRAMSTATE; // Value of P_enumProgramState
	
	bRouterBusy: BOOL; // TRUE while M_RouterHelper is being used by a method

	bTemplateBusy: BOOL;
	bConnectBusy: BOOL;
	bDisconnectBusy: BOOL;
	bGetConnectStatusBusy: BOOL;
	bEnableBusy: BOOL;
	bDisableBusy: BOOL;
	bGetEnableStatusBusy: BOOL;
	bPowerOnBusy: BOOL;
	bPowerOffBusy: BOOL;
	bGetPowerStatusBusy: BOOL;
	bGetCurrentProgramBusy: BOOL;
	bGetProgramStateBusy: BOOL;
	bLoadProgramBusy: BOOL;
	bPauseProgramBusy: BOOL;
	bStartProgramBusy: BOOL;
	bStopProgramBusy: BOOL;
	bResetBusy: BOOL;
	bAbortBusy: BOOL;
	bRouterHelperBusy: BOOL;
	
	intTemplateStep: INT;
	intConnectStep: INT;
	intDisconnectStep: INT;
	intGetConnectStatusStep: INT;
	intEnableStep: INT;
	intDisableStep: INT;
	intGetEnableStatusStep: INT;
	intPowerOnStep: INT;
	intPowerOffStep: INT;
	intGetCurrentProgramStep: INT;
	intGetProgramStateStep: INT;
	intLoadProgramStep: INT;
	intPauseProgramStep: INT;
	intStartProgramStep: INT;
	intStopProgramStep: INT;
	intResetStep: INT;
	intAbortStep: INT;
	intGetPowerStatusStep: INT;
	intRouterHelperStep: INT;
	bTriggerBusy: BOOL;
	intTriggerStep: INT;
END_VAR

A_CommandRecovery();

(* This method should establish any external connections required to use the
	functions of the device, and return TRUE and set P_bConnected to TRUE once
	connected. *)
METHOD M_Abort : BOOL
VAR CONSTANT
	_strCOMMAND_NAME : T_MaxString	:= 'Abort'; // Name of the API method
	_timeCOMMAND_TIMEOUT : TIME		:= T#30S; // Max time to receive API response
	_strSTART_MSG : T_MaxString		:= 'Aborting'; // Prints when method starts
	_strEND_MSG : T_MaxString		:= 'Aborted'; // Prints when method finishes
	_udintERROR_ID : UDINT			:= E_ApiDeviceError.FailedToAbort; // Error ID to set if command fails
	_strERROR_MSG : T_MaxString		:= 'Abort failed!'; // Error message to set if command fails
END_VAR
VAR_INST
	_inst_arrParams: T_ApiParameterList; // Parameters array
	_inst_arrOutputs: T_ApiParameterList; // Outputs array
	_inst_strRet: T_ApiParamValue; // Return string from the router
	_inst_intStep: INT; // Current method step
	_inst_fbParams: FB_ApiParamBuilder; // Parameter builder FB
END_VAR
VAR
	_bComplete: BOOL; // True if the routing finishes
	_intRet: INT; // Return string converted to an integer
	_bResult : BOOL; // Output of the method
	_pArgs: PVOID; // Arguments pointer
END_VAR
_bResult := FALSE;

// Recover from premature stop
bAbortBusy := TRUE;
_inst_intStep := intAbortStep;

// Steps
CASE _inst_intStep OF
	0: // Wait for no error and router not busy
		IF NOT THIS^.P_bError AND NOT bRouterBusy THEN
			bRouterBusy := TRUE;
			_inst_intStep := _inst_intStep + 10;
		END_IF
		
	10: // Initialize parameters
		THIS^.M_LogMessage(_strSTART_MSG);
		_inst_fbParams.M_ClearParameters();
		_pArgs := _inst_fbParams.M_AddEmptyStruct('args');
		_inst_fbParams.M_OutputToParameterList(_inst_arrParams);
		_inst_intStep := _inst_intStep + 10;
		
	20: // Route the command
		_bComplete := M_RouterHelper(
			_in_strMethodName := _strCOMMAND_NAME, 
			_in_timeTimeout := _timeCOMMAND_TIMEOUT,
			_inout_arrParams := _inst_arrParams,
			_inout_arrOutputs := _inst_arrOutputs,
			_out_strReturnValue=>_inst_strRet);
		
		// If route completed, move to next step
		IF _bComplete THEN
			_inst_intStep := _inst_intStep + 10;
			bRouterBusy := FALSE;
		ELSIF THIS^.P_bError THEN
			_inst_intStep := 0;
			bRouterBusy := FALSE;
		END_IF
		
	30: // Parse results
		_intRet := STRING_TO_INT(_inst_strRet);
		IF _intRet > 0 THEN
			_bResult := TRUE;
			THIS^.M_LogMessage(_strEND_MSG);
			_inst_fbParams.M_LoadFromParameterList(_inst_arrOutputs);
			
		// Set error if command failed
		ELSE
			THIS^.M_SetError(_udintERROR_ID, _strERROR_MSG);
		END_IF
		
		// Go back to start
		_inst_intStep := 0;
END_CASE

M_Abort := _bResult;
intAbortStep := _inst_intStep;
END_METHOD

(* This property should be TRUE while any method in this interface is actively
	executing, or FALSE otherwise. *)
PROPERTY P_bAbortBusy : BOOL
GET
P_bAbortBusy := bRouterBusy;
END_GET
END_PROPERTY

(* This method should establish any external connections required to use the
	functions of the device, and return TRUE and set P_bConnected to TRUE once
	connected. *)
METHOD M_Connect : BOOL
VAR CONSTANT
	_strCOMMAND_NAME : T_MaxString	:= 'Connect'; // Name of the API method
	_timeCOMMAND_TIMEOUT : TIME		:= T#30S; // Max time to receive API response
	_strSTART_MSG : T_MaxString		:= 'Connecting'; // Prints when method starts
	_strEND_MSG : T_MaxString		:= 'Connected'; // Prints when method finishes
	_udintERROR_ID : UDINT			:= E_ApiDeviceError.FailedToConnect; // Error ID to set if command fails
	_strERROR_MSG : T_MaxString		:= 'Failed to connect!'; // Error message to set if command fails
END_VAR
VAR_INST
	_inst_arrParams: T_ApiParameterList; // Parameters array
	_inst_arrOutputs: T_ApiParameterList; // Outputs array
	_inst_strRet: T_ApiParamValue; // Return string from the router
	_inst_intStep: INT; // Current method step
	_inst_fbParams: FB_ApiParamBuilder; // Parameter builder FB
END_VAR
VAR
	_bComplete: BOOL; // True if the routing finishes
	_intRet: INT; // Return string converted to an integer
	_bResult : BOOL; // Output of the method
	_pArgs: PVOID; // Arguments pointer
END_VAR
_bResult := FALSE;

// Recover from premature stop
bConnectBusy := TRUE;
_inst_intStep := intConnectStep;

// Steps
CASE _inst_intStep OF
	0: // Wait for no error and router not busy
		IF NOT THIS^.P_bError AND NOT bRouterBusy THEN
			bRouterBusy := TRUE;
			_inst_intStep := _inst_intStep + 10;
		END_IF
		
	10: // Initialize parameters
		THIS^.M_LogMessage(_strSTART_MSG);
		_inst_fbParams.M_ClearParameters();
		_pArgs := _inst_fbParams.M_AddEmptyStruct('args');
		_inst_fbParams.M_OutputToParameterList(_inst_arrParams);
		_inst_intStep := _inst_intStep + 10;
		
	20: // Route the command
		_bComplete := M_RouterHelper(
			_in_strMethodName := _strCOMMAND_NAME, 
			_in_timeTimeout := _timeCOMMAND_TIMEOUT,
			_inout_arrParams := _inst_arrParams,
			_inout_arrOutputs := _inst_arrOutputs,
			_out_strReturnValue=>_inst_strRet);
		
		// If route completed, move to next step
		IF _bComplete THEN
			_inst_intStep := _inst_intStep + 10;
			bRouterBusy := FALSE;
		ELSIF THIS^.P_bError THEN
			_inst_intStep := 0;
			bRouterBusy := FALSE;
		END_IF
		
	30: // Parse results
		_intRet := STRING_TO_INT(_inst_strRet);
		IF _intRet > 0 THEN
			_bResult := TRUE;
			THIS^.M_LogMessage(_strEND_MSG);
			_inst_fbParams.M_LoadFromParameterList(_inst_arrOutputs);
			bConnected := TRUE;
			
		// Set error if command failed
		ELSE
			THIS^.M_SetError(_udintERROR_ID, _strERROR_MSG);
		END_IF
		
		// Go back to start
		_inst_intStep := 0;
END_CASE

M_Connect := _bResult;
intConnectStep := _inst_intStep;
END_METHOD

(* This method should break any connections established by M_Connect. It should
	immediately set P_bConnected to false unless all connections are known to
	be still active, and return TRUE once those connections are all fully
	disconnected. *)
METHOD M_Disconnect : BOOL
VAR CONSTANT
	_strCOMMAND_NAME : T_MaxString	:= 'Disconnect'; // Name of the API method
	_timeCOMMAND_TIMEOUT : TIME		:= T#30S; // Max time to receive API response
	_strSTART_MSG : T_MaxString		:= 'Disconnecting'; // Prints when method starts
	_strEND_MSG : T_MaxString		:= 'Disconnected'; // Prints when method finishes
	_udintERROR_ID : UDINT			:= E_ApiDeviceError.FailedToDisconnect; // Error ID to set if command fails
	_strERROR_MSG : T_MaxString		:= 'Failed to disconnect!'; // Error message to set if command fails
END_VAR
VAR_INST
	_inst_arrParams: T_ApiParameterList; // Parameters array
	_inst_arrOutputs: T_ApiParameterList; // Outputs array
	_inst_strRet: T_ApiParamValue; // Return string from the router
	_inst_intStep: INT; // Current method step
	_inst_fbParams: FB_ApiParamBuilder; // Parameter builder FB
END_VAR
VAR
	_bComplete: BOOL; // True if the routing finishes
	_intRet: INT; // Return string converted to an integer
	_bResult : BOOL; // Output of the method
	_pArgs: PVOID; // Arguments pointer
END_VAR
_bResult := FALSE;

// Recover from premature stop
bDisconnectBusy := TRUE;
_inst_intStep := intDisconnectStep;

// Steps
CASE _inst_intStep OF
	0: // Wait for no error and router not busy
		IF NOT THIS^.P_bError AND NOT bRouterBusy THEN
			bRouterBusy := TRUE;
			_inst_intStep := _inst_intStep + 10;
		END_IF
		
	10: // Initialize parameters
		THIS^.M_LogMessage(_strSTART_MSG);
		_inst_fbParams.M_ClearParameters();
		_pArgs := _inst_fbParams.M_AddEmptyStruct('args');
		_inst_fbParams.M_OutputToParameterList(_inst_arrParams);
		_inst_intStep := _inst_intStep + 10;
		
	20: // Route the command
		_bComplete := M_RouterHelper(
			_in_strMethodName := _strCOMMAND_NAME, 
			_in_timeTimeout := _timeCOMMAND_TIMEOUT,
			_inout_arrParams := _inst_arrParams,
			_inout_arrOutputs := _inst_arrOutputs,
			_out_strReturnValue=>_inst_strRet);
		
		// If route completed, move to next step
		IF _bComplete THEN
			_inst_intStep := _inst_intStep + 10;
			bRouterBusy := FALSE;
		ELSIF THIS^.P_bError THEN
			_inst_intStep := 0;
			bRouterBusy := FALSE;
		END_IF
		
	30: // Parse results
		_intRet := STRING_TO_INT(_inst_strRet);
		IF _intRet > 0 THEN
			_bResult := TRUE;
			THIS^.M_LogMessage(_strEND_MSG);
			_inst_fbParams.M_LoadFromParameterList(_inst_arrOutputs);
			bConnected := FALSE;
			
		// Set error if command failed
		ELSE
			THIS^.M_SetError(_udintERROR_ID, _strERROR_MSG);
		END_IF
		
		// Go back to start
		_inst_intStep := 0;
END_CASE

M_Disconnect := _bResult;
intDisconnectStep := _inst_intStep;
END_METHOD

(* This method should explicitly check the connection status of the device.
	Once the connection status is known, this method should return TRUE.
	If this method fails, P_bConnected should be set to FALSE since the device
	is not absolutely known to still be connected. *)
METHOD M_GetConnectStatus : BOOL
VAR_OUTPUT
	(* This should return TRUE if all connections required to make the device
		function properly are known to be connected, and FALSE otherwise. *)
	bConnected	: BOOL;
END_VAR
VAR CONSTANT
	_strCOMMAND_NAME : T_MaxString	:= 'GetConnectStatus'; // Name of the API method
	_timeCOMMAND_TIMEOUT : TIME		:= T#5S; // Max time to receive API response
	_strSTART_MSG : T_MaxString		:= 'Getting connection status'; // Prints when method starts
	_strEND_MSG : T_MaxString		:= 'Received connection status'; // Prints when method finishes
	_udintERROR_ID : UDINT			:= E_ApiDeviceError.FailedToGetConnectStatus; // Error ID to set if command fails
	_strERROR_MSG : T_MaxString		:= 'Failed to get connection status!'; // Error message to set if command fails
END_VAR
VAR_INST
	_inst_arrParams: T_ApiParameterList; // Parameters array
	_inst_arrOutputs: T_ApiParameterList; // Outputs array
	_inst_strRet: T_ApiParamValue; // Return string from the router
	_inst_intStep: INT; // Current method step
	_inst_fbParams: FB_ApiParamBuilder; // Parameter builder FB
END_VAR
VAR
	_bComplete: BOOL; // True if the routing finishes
	_intRet: INT; // Return string converted to an integer
	_bResult : BOOL; // Output of the method
	_pArgs: PVOID; // Arguments pointer
END_VAR
_bResult := FALSE;

// Recover from premature stop
bGetConnectStatusBusy := TRUE;
_inst_intStep := intGetConnectStatusStep;

// Steps
CASE _inst_intStep OF
	0: // Wait for no error and router not busy
		IF NOT THIS^.P_bError AND NOT bRouterBusy THEN
			bRouterBusy := TRUE;
			_inst_intStep := _inst_intStep + 10;
		END_IF
		
	10: // Initialize parameters
		THIS^.M_LogMessage(_strSTART_MSG);
		_inst_fbParams.M_ClearParameters();
		_pArgs := _inst_fbParams.M_AddEmptyStruct('args');
		_inst_fbParams.M_OutputToParameterList(_inst_arrParams);
		_inst_intStep := _inst_intStep + 10;
		
	20: // Route the command
		_bComplete := M_RouterHelper(
			_in_strMethodName := _strCOMMAND_NAME, 
			_in_timeTimeout := _timeCOMMAND_TIMEOUT,
			_inout_arrParams := _inst_arrParams,
			_inout_arrOutputs := _inst_arrOutputs,
			_out_strReturnValue=>_inst_strRet);
		
		// If route completed, move to next step
		IF _bComplete THEN
			_inst_intStep := _inst_intStep + 10;
			bRouterBusy := FALSE;
		ELSIF THIS^.P_bError THEN
			_inst_intStep := 0;
			bRouterBusy := FALSE;
		END_IF
		
	30: // Parse results
		_intRet := STRING_TO_INT(_inst_strRet);
		IF _intRet > 0 THEN
			_bResult := TRUE;
			THIS^.M_LogMessage(_strEND_MSG);
			_inst_fbParams.M_LoadFromParameterList(_inst_arrOutputs);
			THIS^.bConnected := _inst_fbParams.M_ParseBool(
				_inst_fbParams.M_GetParameter('connected'));
			bConnected := THIS^.bConnected;
			
		// Set error if command failed
		ELSE
			THIS^.M_SetError(_udintERROR_ID, _strERROR_MSG);
		END_IF
		
		// Go back to start
		_inst_intStep := 0;
END_CASE

M_GetConnectStatus := _bResult;
intGetConnectStatusStep := _inst_intStep;
END_METHOD

(* This property should be TRUE while any method in this interface is actively
	executing, or FALSE otherwise. *)
PROPERTY P_bConnectBusy : BOOL
GET
P_bConnectBusy := bRouterBusy;
END_GET
END_PROPERTY

(* This should be set to TRUE if M_Connect is successful or M_GetConnectStatus
	determines the device to be connected, and set to FALSE if M_Disconnect is
	called at all, M_GetConnectStatus fails, or M_GetConnectStatus determines
	the device to be not connected. *)
PROPERTY P_bConnected : BOOL
GET
P_bConnected := bConnected;
END_GET
END_PROPERTY

(* This method should return to the device to the state it was prior to being
	enabled. P_bEnabled should be immediately set to false unless the status of
	the device is explicitly known to still be enabled. After being disabled,
	the device should typically be unable to perform process steps. Once
	successfully disabled, this method should return TRUE. *)
METHOD M_Disable : BOOL
VAR CONSTANT
	_strCOMMAND_NAME : T_MaxString	:= 'Disable'; // Name of the API method
	_timeCOMMAND_TIMEOUT : TIME		:= T#30S; // Max time to receive API response
	_strSTART_MSG : T_MaxString		:= 'Disabling'; // Prints when method starts
	_strEND_MSG : T_MaxString		:= 'Disabled'; // Prints when method finishes
	_udintERROR_ID : UDINT			:= E_ApiDeviceError.FailedToDisable; // Error ID to set if command fails
	_strERROR_MSG : T_MaxString		:= 'Failed to disable!'; // Error message to set if command fails
END_VAR
VAR_INST
	_inst_arrParams: T_ApiParameterList; // Parameters array
	_inst_arrOutputs: T_ApiParameterList; // Outputs array
	_inst_strRet: T_ApiParamValue; // Return string from the router
	_inst_intStep: INT; // Current method step
	_inst_fbParams: FB_ApiParamBuilder; // Parameter builder FB
END_VAR
VAR
	_bComplete: BOOL; // True if the routing finishes
	_intRet: INT; // Return string converted to an integer
	_bResult : BOOL; // Output of the method
	_pArgs: PVOID; // Arguments pointer
END_VAR
_bResult := FALSE;

// Recover from premature stop
bDisableBusy := TRUE;
_inst_intStep := intDisableStep;

// Steps
CASE _inst_intStep OF
	0: // Wait for no error and router not busy
		IF NOT THIS^.P_bError AND NOT bRouterBusy THEN
			bRouterBusy := TRUE;
			_inst_intStep := _inst_intStep + 10;
		END_IF
		
	10: // Initialize parameters
		THIS^.M_LogMessage(_strSTART_MSG);
		_inst_fbParams.M_ClearParameters();
		_pArgs := _inst_fbParams.M_AddEmptyStruct('args');
		_inst_fbParams.M_OutputToParameterList(_inst_arrParams);
		_inst_intStep := _inst_intStep + 10;
		
	20: // Route the command
		_bComplete := M_RouterHelper(
			_in_strMethodName := _strCOMMAND_NAME, 
			_in_timeTimeout := _timeCOMMAND_TIMEOUT,
			_inout_arrParams := _inst_arrParams,
			_inout_arrOutputs := _inst_arrOutputs,
			_out_strReturnValue=>_inst_strRet);
		
		// If route completed, move to next step
		IF _bComplete THEN
			_inst_intStep := _inst_intStep + 10;
			bRouterBusy := FALSE;
		ELSIF THIS^.P_bError THEN
			_inst_intStep := 0;
			bRouterBusy := FALSE;
		END_IF
		
	30: // Parse results
		_intRet := STRING_TO_INT(_inst_strRet);
		IF _intRet > 0 THEN
			_bResult := TRUE;
			THIS^.M_LogMessage(_strEND_MSG);
			_inst_fbParams.M_LoadFromParameterList(_inst_arrOutputs);
			bEnabled := FALSE;
			
		// Set error if command failed
		ELSE
			THIS^.M_SetError(_udintERROR_ID, _strERROR_MSG);
		END_IF
		
		// Go back to start
		_inst_intStep := 0;
END_CASE

M_Disable := _bResult;
intDisableStep := _inst_intStep;
END_METHOD

(* This method should perform any tasks that must be performed after a device
	is energized, but prior to the device being used in a process, and then
	return TRUE and set P_bEnabled to TRUE once those tasks are completed. *)
METHOD M_Enable : BOOL
VAR CONSTANT
	_strCOMMAND_NAME : T_MaxString	:= 'Enable'; // Name of the API method
	_timeCOMMAND_TIMEOUT : TIME		:= T#30S; // Max time to receive API response
	_strSTART_MSG : T_MaxString		:= 'Enabling'; // Prints when method starts
	_strEND_MSG : T_MaxString		:= 'Enabled'; // Prints when method finishes
	_udintERROR_ID : UDINT			:= E_ApiDeviceError.FailedToEnable; // Error ID to set if command fails
	_strERROR_MSG : T_MaxString		:= 'Failed to enable!'; // Error message to set if command fails
END_VAR
VAR_INST
	_inst_arrParams: T_ApiParameterList; // Parameters array
	_inst_arrOutputs: T_ApiParameterList; // Outputs array
	_inst_strRet: T_ApiParamValue; // Return string from the router
	_inst_intStep: INT; // Current method step
	_inst_fbParams: FB_ApiParamBuilder; // Parameter builder FB
END_VAR
VAR
	_bComplete: BOOL; // True if the routing finishes
	_intRet: INT; // Return string converted to an integer
	_bResult : BOOL; // Output of the method
	_pArgs: PVOID; // Arguments pointer
END_VAR
_bResult := FALSE;

// Recover from premature stop
bEnableBusy := TRUE;
_inst_intStep := intEnableStep;

// Steps
CASE _inst_intStep OF
	0: // Wait for no error and router not busy
		IF NOT THIS^.P_bError AND NOT bRouterBusy THEN
			bRouterBusy := TRUE;
			_inst_intStep := _inst_intStep + 10;
		END_IF
		
	10: // Initialize parameters
		THIS^.M_LogMessage(_strSTART_MSG);
		_inst_fbParams.M_ClearParameters();
		_pArgs := _inst_fbParams.M_AddEmptyStruct('args');
		_inst_fbParams.M_OutputToParameterList(_inst_arrParams);
		_inst_intStep := _inst_intStep + 10;
		
	20: // Route the command
		_bComplete := M_RouterHelper(
			_in_strMethodName := _strCOMMAND_NAME, 
			_in_timeTimeout := _timeCOMMAND_TIMEOUT,
			_inout_arrParams := _inst_arrParams,
			_inout_arrOutputs := _inst_arrOutputs,
			_out_strReturnValue=>_inst_strRet);
		
		// If route completed, move to next step
		IF _bComplete THEN
			_inst_intStep := _inst_intStep + 10;
			bRouterBusy := FALSE;
		ELSIF THIS^.P_bError THEN
			_inst_intStep := 0;
			bRouterBusy := FALSE;
		END_IF
		
	30: // Parse results
		_intRet := STRING_TO_INT(_inst_strRet);
		IF _intRet > 0 THEN
			_bResult := TRUE;
			THIS^.M_LogMessage(_strEND_MSG);
			_inst_fbParams.M_LoadFromParameterList(_inst_arrOutputs);
			bEnabled := TRUE;
			
		// Set error if command failed
		ELSE
			THIS^.M_SetError(_udintERROR_ID, _strERROR_MSG);
		END_IF
		
